gfCNCPoint2[16840] = {X 155.3044, Y 59.7694, Z -3.0000, A 0.000, B 0.000, C 0.000 }
gfCNCPoint2[16841] = {X 155.2181, Y 58.9678, Z -3.0000, A 0.000, B 0.000, C 0.000 }
gfCNCPoint2[16842] = {X 155.2180, Y 58.0000, Z -3.0000, A 0.000, B 0.000, C 0.000 }
gfCNCPoint2[16843] = {X 155.3203, Y 57.0921, Z -3.0000, A 0.000, B 0.000, C 0.000 }
gfCNCPoint2[16844] = {X 155.6220, Y 56.2298, Z -3.0000, A 0.000, B 0.000, C 0.000 }
gfCNCPoint2[16845] = {X 156.1081, Y 55.4562, Z -3.0000, A 0.000, B 0.000, C 0.000 }
gfCNCPoint2[16846] = {X 156.7541, Y 54.8101, Z -3.0000, A 0.000, B 0.000, C 0.000 }
gfCNCPoint2[16847] = {X 157.5277, Y 54.3240, Z -3.0000, A 0.000, B 0.000, C 0.000 }
gfCNCPoint2[16848] = {X 158.3901, Y 54.0223, Z -3.0000, A 0.000, B 0.000, C 0.000 }
gfCNCPoint2[16849] = {X 159.2980, Y 53.9200, Z -3.0000, A 0.000, B 0.000, C 0.000 }
gfCNCPoint2[16850] = {X 178.5335, Y 53.9200, Z -3.0000, A 0.000, B 0.000, C 0.000 }
gfCNCPoint2[16851] = {X 179.4414, Y 54.0223, Z -3.0000, A 0.000, B 0.000, C 0.000 }
gfCNCPoint2[16852] = {X 180.3037, Y 54.3240, Z -3.0000, A 0.000, B 0.000, C 0.000 }
gfCNCPoint2[16853] = {X 181.0773, Y 54.8101, Z -3.0000, A 0.000, B 0.000, C 0.000 }
gfCNCPoint2[16854] = {X 181.7234, Y 55.4562, Z -3.0000, A 0.000, B 0.000, C 0.000 }
gfCNCPoint2[16855] = {X 182.2095, Y 56.2298, Z -3.0000, A 0.000, B 0.000, C 0.000 }
gfCNCPoint2[16856] = {X 182.5112, Y 57.0921, Z -3.0000, A 0.000, B 0.000, C 0.000 }
gfCNCPoint2[16857] = {X 182.6135, Y 58.0000, Z -3.0000, A 0.000, B 0.000, C 0.000 }
gfCNCPoint2[16858] = {X 182.6135, Y 58.9342, Z -3.0000, A 0.000, B 0.000, C 0.000 }
gfCNCPoint2[16859] = {X 182.5334, Y 59.7385, Z -3.0000, A 0.000, B 0.000, C 0.000 }
gfCNCPoint2[16860] = {X 182.2963, Y 60.5113, Z -3.0000, A 0.000, B 0.000, C 0.000 }
gfCNCPoint2[16861] = {X 181.9116, Y 61.2221, Z -3.0000, A 0.000, B 0.000, C 0.000 }
gfCNCPoint2[16862] = {X 209.3010, Y 91.1161, Z -3.0000, A 0.000, B 0.000, C 0.000 }
gfCNCPoint2[16863] = {X 209.9711, Y 91.7959, Z -3.0000, A 0.000, B 0.000, C 0.000 }
gfCNCPoint2[16864] = {X 210.6888, Y 92.4252, Z -3.0000, A 0.000, B 0.000, C 0.000 }
gfCNCPoint2[16865] = {X 211.0137, Y 92.6303, Z -3.0000, A 0.000, B 0.000, C 0.000 }
gfCNCPoint2[16866] = {X 211.3781, Y 92.7521, Z -3.0000, A 0.000, B 0.000, C 0.000 }
gfCNCPoint2[16867] = {X 213.3970, Y 93.0670, Z -3.0000, A 0.000, B 0.000, C 0.000 }
gfCNCPoint2[16868] = {X 214.4547, Y 92.9770, Z -3.0000, A 0.000, B 0.000, C 0.000 }
gfCNCPoint2[16869] = {X 215.5145, Y 92.9161, Z -3.0000, A 0.000, B 0.000, C 0.000 }
gfCNCPoint2[16870] = {X 216.2276, Y 92.8376, Z -3.0000, A 0.000, B 0.000, C 0.000 }
gfCNCPoint2[16871] = {X 216.9142, Y 92.6297, Z -3.0000, A 0.000, B 0.000, C 0.000 }
gfCNCPoint2[16872] = {X 217.5510, Y 92.2995, Z -3.0000, A 0.000, B 0.000, C 0.000 }
gfCNCPoint2[16873] = {X 223.0910, Y 88.7242, Z -3.0000, A 0.000, B 0.000, C 0.000 }
gfCNCPoint2[16874] = {X 246.3547, Y 73.8481, Z -3.0000, A 0.000, B 0.000, C 0.000 }
gfCNCPoint2[16875] = {X 221.7196, Y 64.1802, Z -3.0000, A 0.000, B 0.000, C 0.000 }
gfCNCPoint2[16876] = {X 219.9262, Y 63.5800, Z -3.0000, A 0.000, B 0.000, C 0.000 }
gfCNCPoint2[16877] = {X 218.0758, Y 63.1888, Z -3.0000, A 0.000, B 0.000, C 0.000 }
gfCNCPoint2[16878] = {X 216.1929, Y 63.0117, Z -3.0000, A 0.000, B 0.000, C 0.000 }
gfCNCPoint2[16879] = {X 215.3127, Y 62.8850, Z -3.0000, A 0.000, B 0.000, C 0.000 }
gfCNCPoint2[16880] = {X 214.4809, Y 62.5706, Z -3.0000, A 0.000, B 0.000, C 0.000 }
gfCNCPoint2[16881] = {X 213.7370, Y 62.0834, Z -3.0000, A 0.000, B 0.000, C 0.000 }
gfCNCPoint2[16882] = {X 213.1162, Y 61.4466, Z -3.0000, A 0.000, B 0.000, C 0.000 }
gfCNCPoint2[16883] = {X 212.6482, Y 60.6905, Z -3.0000, A 0.000, B 0.000, C 0.000 }
gfCNCPoint2[16884] = {X 212.3552, Y 59.8509, Z -3.0000, A 0.000, B 0.000, C 0.000 }
gfCNCPoint2[16885] = {X 212.2509, Y 58.9678, Z -3.0000, A 0.000, B 0.000, C 0.000 }
gfCNCPoint2[16886] = {X 212.2508, Y 58.0000, Z -3.0000, A 0.000, B 0.000, C 0.000 }
gfCNCPoint2[16887] = {X 212.3531, Y 57.0921, Z -3.0000, A 0.000, B 0.000, C 0.000 }
gfCNCPoint2[16888] = {X 212.6549, Y 56.2298, Z -3.0000, A 0.000, B 0.000, C 0.000 }
gfCNCPoint2[16889] = {X 213.1409, Y 55.4562, Z -3.0000, A 0.000, B 0.000, C 0.000 }
gfCNCPoint2[16890] = {X 213.7870, Y 54.8101, Z -3.0000, A 0.000, B 0.000, C 0.000 }
gfCNCPoint2[16891] = {X 214.5606, Y 54.3240, Z -3.0000, A 0.000, B 0.000, C 0.000 }
gfCNCPoint2[16892] = {X 215.4229, Y 54.0223, Z -3.0000, A 0.000, B 0.000, C 0.000 }
gfCNCPoint2[16893] = {X 216.3308, Y 53.9200, Z -3.0000, A 0.000, B 0.000, C 0.000 }
gfCNCPoint2[16894] = {X 237.2617, Y 53.9200, Z -3.0000, A 0.000, B 0.000, C 0.000 }
gfCNCPoint2[16895] = {X 238.1696, Y 54.0223, Z -3.0000, A 0.000, B 0.000, C 0.000 }
gfCNCPoint2[16896] = {X 239.0319, Y 54.3240, Z -3.0000, A 0.000, B 0.000, C 0.000 }
gfCNCPoint2[16897] = {X 239.8055, Y 54.8101, Z -3.0000, A 0.000, B 0.000, C 0.000 }
gfCNCPoint2[16898] = {X 240.4516, Y 55.4562, Z -3.0000, A 0.000, B 0.000, C 0.000 }
gfCNCPoint2[16899] = {X 240.9376, Y 56.2298, Z -3.0000, A 0.000, B 0.000, C 0.000 }
gfCNCPoint2[16900] = {X 241.2394, Y 57.0921, Z -3.0000, A 0.000, B 0.000, C 0.000 }
gfCNCPoint2[16901] = {X 241.3417, Y 58.0000, Z -3.0000, A 0.000, B 0.000, C 0.000 }
gfCNCPoint2[16902] = {X 241.3417, Y 58.3967, Z -3.0000, A 0.000, B 0.000, C 0.000 }
gfCNCPoint2[16903] = {X 247.4005, Y 60.7586, Z -3.0000, A 0.000, B 0.000, C 0.000 }
gfCNCPoint2[16904] = {X 275.8735, Y 72.0561, Z -3.0000, A 0.000, B 0.000, C 0.000 }
gfCNCPoint2[16905] = {X 275.8743, Y 62.9983, Z -3.0000, A 0.000, B 0.000, C 0.000 }
gfCNCPoint2[16906] = {X 275.7380, Y 62.9840, Z -3.0000, A 0.000, B 0.000, C 0.000 }
gfCNCPoint2[16907] = {X 275.6022, Y 62.9651, Z -3.0000, A 0.000, B 0.000, C 0.000 }
gfCNCPoint2[16908] = {X 274.6826, Y 62.7081, Z -3.0000, A 0.000, B 0.000, C 0.000 }
gfCNCPoint2[16909] = {X 273.8479, Y 62.2445, Z -3.0000, A 0.000, B 0.000, C 0.000 }
gfCNCPoint2[16910] = {X 273.1438, Y 61.5996, Z -3.0000, A 0.000, B 0.000, C 0.000 }
gfCNCPoint2[16911] = {X 272.6088, Y 60.8087, Z -3.0000, A 0.000, B 0.000, C 0.000 }
gfCNCPoint2[16912] = {X 272.2724, Y 59.9151, Z -3.0000, A 0.000, B 0.000, C 0.000 }
gfCNCPoint2[16913] = {X 272.1528, Y 58.9678, Z -3.0000, A 0.000, B 0.000, C 0.000 }
gfCNCPoint2[16914] = {X 272.1527, Y 58.0000, Z -3.0000, A 0.000, B 0.000, C 0.000 }
gfCNCPoint2[16915] = {X 272.2550, Y 57.0921, Z -3.0000, A 0.000, B 0.000, C 0.000 }
gfCNCPoint2[16916] = {X 272.5567, Y 56.2298, Z -3.0000, A 0.000, B 0.000, C 0.000 }
gfCNCPoint2[16917] = {X 273.0428, Y 55.4562, Z -3.0000, A 0.000, B 0.000, C 0.000 }
gfCNCPoint2[16918] = {X 273.6889, Y 54.8101, Z -3.0000, A 0.000, B 0.000, C 0.000 }
gfCNCPoint2[16919] = {X 274.4624, Y 54.3240, Z -3.0000, A 0.000, B 0.000, C 0.000 }
gfCNCPoint2[16920] = {X 275.3248, Y 54.0223, Z -3.0000, A 0.000, B 0.000, C 0.000 }
gfCNCPoint2[16921] = {X 276.2327, Y 53.9200, Z -3.0000, A 0.000, B 0.000, C 0.000 }
gfCNCPoint2[16922] = {X 292.7731, Y 53.9200, Z -3.0000, A 0.000, B 0.000, C 0.000 }
gfCNCPoint2[16923] = {X 293.6810, Y 54.0223, Z -3.0000, A 0.000, B 0.000, C 0.000 }
gfCNCPoint2[16924] = {X 294.5433, Y 54.3240, Z -3.0000, A 0.000, B 0.000, C 0.000 }
gfCNCPoint2[16925] = {X 295.3169, Y 54.8101, Z -3.0000, A 0.000, B 0.000, C 0.000 }
gfCNCPoint2[16926] = {X 295.9630, Y 55.4562, Z -3.0000, A 0.000, B 0.000, C 0.000 }
gfCNCPoint2[16927] = {X 296.4490, Y 56.2298, Z -3.0000, A 0.000, B 0.000, C 0.000 }
gfCNCPoint2[16928] = {X 296.7508, Y 57.0921, Z -3.0000, A 0.000, B 0.000, C 0.000 }
gfCNCPoint2[16929] = {X 296.8531, Y 58.0000, Z -3.0000, A 0.000, B 0.000, C 0.000 }
gfCNCPoint2[16930] = {X 296.8531, Y 58.9344, Z -3.0000, A 0.000, B 0.000, C 0.000 }
gfCNCPoint2[16931] = {X 296.7374, Y 59.8874, Z -3.0000, A 0.000, B 0.000, C 0.000 }
gfCNCPoint2[16932] = {X 296.4031, Y 60.7873, Z -3.0000, A 0.000, B 0.000, C 0.000 }
gfCNCPoint2[16933] = {X 295.8686, Y 61.5848, Z -3.0000, A 0.000, B 0.000, C 0.000 }
gfCNCPoint2[16934] = {X 295.1631, Y 62.2359, Z -3.0000, A 0.000, B 0.000, C 0.000 }
gfCNCPoint2[16935] = {X 294.3255, Y 62.7050, Z -3.0000, A 0.000, B 0.000, C 0.000 }
gfCNCPoint2[16936] = {X 293.4017, Y 62.9663, Z -3.0000, A 0.000, B 0.000, C 0.000 }
gfCNCPoint2[16937] = {X 293.2752, Y 62.9845, Z -3.0000, A 0.000, B 0.000, C 0.000 }
gfCNCPoint2[16938] = {X 293.1481, Y 62.9987, Z -3.0000, A 0.000, B 0.000, C 0.000 }
gfCNCPoint2[16939] = {X 293.1321, Y 63.1581, Z -3.0000, A 0.000, B 0.000, C 0.000 }
gfCNCPoint2[16940] = {X 293.1443, Y 92.9938, Z -3.0000, A 0.000, B 0.000, C 0.000 }
gfCNCPoint2[16941] = {X 293.2728, Y 93.0085, Z -3.0000, A 0.000, B 0.000, C 0.000 }
gfCNCPoint2[16942] = {X 293.4007, Y 93.0272, Z -3.0000, A 0.000, B 0.000, C 0.000 }
gfCNCPoint2[16943] = {X 294.3242, Y 93.2911, Z -3.0000, A 0.000, B 0.000, C 0.000 }
gfCNCPoint2[16944] = {X 295.1614, Y 93.7620, Z -3.0000, A 0.000, B 0.000, C 0.000 }
gfCNCPoint2[16945] = {X 295.8665, Y 94.4142, Z -3.0000, A 0.000, B 0.000, C 0.000 }
gfCNCPoint2[16946] = {X 296.4011, Y 95.2122, Z -3.0000, A 0.000, B 0.000, C 0.000 }
gfCNCPoint2[16947] = {X 296.7360, Y 96.1124, Z -3.0000, A 0.000, B 0.000, C 0.000 }
gfCNCPoint2[16948] = {X 296.8531, Y 97.0657, Z -3.0000, A 0.000, B 0.000, C 0.000 }
gfCNCPoint2[16949] = {X 296.8531, Y 98.0000, Z -3.0000, A 0.000, B 0.000, C 0.000 }
gfCNCPoint2[16950] = {X 296.7508, Y 98.9079, Z -3.0000, A 0.000, B 0.000, C 0.000 }
gfCNCPoint2[16951] = {X 296.4490, Y 99.7702, Z -3.0000, A 0.000, B 0.000, C 0.000 }
gfCNCPoint2[16952] = {X 295.9630, Y 100.5438, Z -3.0000, A 0.000, B 0.000, C 0.000 }
gfCNCPoint2[16953] = {X 295.3169, Y 101.1899, Z -3.0000, A 0.000, B 0.000, C 0.000 }
gfCNCPoint2[16954] = {X 294.5433, Y 101.6760, Z -3.0000, A 0.000, B 0.000, C 0.000 }
gfCNCPoint2[16955] = {X 293.6810, Y 101.9777, Z -3.0000, A 0.000, B 0.000, C 0.000 }
gfCNCPoint2[16956] = {X 292.7731, Y 102.0800, Z -3.0000, A 0.000, B 0.000, C 0.000 }
gfCNCPoint2[16957] = {X 276.2327, Y 102.0800, Z -3.0000, A 0.000, B 0.000, C 0.000 }
gfCNCPoint2[16958] = {X 275.3248, Y 101.9777, Z -3.0000, A 0.000, B 0.000, C 0.000 }
gfCNCPoint2[16959] = {X 274.4624, Y 101.6760, Z -3.0000, A 0.000, B 0.000, C 0.000 }
gfCNCPoint2[16960] = {X 273.6889, Y 101.1899, Z -3.0000, A 0.000, B 0.000, C 0.000 }
gfCNCPoint2[16961] = {X 273.0428, Y 100.5438, Z -3.0000, A 0.000, B 0.000, C 0.000 }
gfCNCPoint2[16962] = {X 272.5567, Y 99.7702, Z -3.0000, A 0.000, B 0.000, C 0.000 }
gfCNCPoint2[16963] = {X 272.2550, Y 98.9079, Z -3.0000, A 0.000, B 0.000, C 0.000 }
gfCNCPoint2[16964] = {X 272.1527, Y 98.0000, Z -3.0000, A 0.000, B 0.000, C 0.000 }
gfCNCPoint2[16965] = {X 272.1527, Y 97.0659, Z -3.0000, A 0.000, B 0.000, C 0.000 }
gfCNCPoint2[16966] = {X 272.2437, Y 96.2088, Z -3.0000, A 0.000, B 0.000, C 0.000 }
gfCNCPoint2[16967] = {X 272.5128, Y 95.3899, Z -3.0000, A 0.000, B 0.000, C 0.000 }
gfCNCPoint2[16968] = {X 272.9480, Y 94.6458, Z -3.0000, A 0.000, B 0.000, C 0.000 }
gfCNCPoint2[16969] = {X 273.5297, Y 94.0097, Z -3.0000, A 0.000, B 0.000, C 0.000 }
gfCNCPoint2[16970] = {X 274.2321, Y 93.5101, Z -3.0000, A 0.000, B 0.000, C 0.000 }
gfCNCPoint2[16971] = {X 275.0238, Y 93.1692, Z -3.0000, A 0.000, B 0.000, C 0.000 }
gfCNCPoint2[16972] = {X 275.8694, Y 93.0021, Z -3.0000, A 0.000, B 0.000, C 0.000 }
gfCNCPoint2[16973] = {X 275.8694, Y 85.4313, Z -3.0000, A 0.000, B 0.000, C 0.000 }
gfCNCPoint2[16974] = {X 262.6143, Y 80.2353, Z -3.0000, A 0.000, B 0.000, C 0.000 }
gfCNCPoint2[16975] = {X 262.1471, Y 80.5294, Z -3.0000, A 0.000, B 0.000, C 0.000 }
gfCNCPoint2[16976] = {X 237.5552, Y 96.4582, Z -3.0000, A 0.000, B 0.000, C 0.000 }
gfCNCPoint2[16977] = {X 237.5598, Y 97.0656, Z -3.0000, A 0.000, B 0.000, C 0.000 }
gfCNCPoint2[16978] = {X 237.5598, Y 98.0000, Z -3.0000, A 0.000, B 0.000, C 0.000 }
gfCNCPoint2[16979] = {X 237.4575, Y 98.9079, Z -3.0000, A 0.000, B 0.000, C 0.000 }
gfCNCPoint2[16980] = {X 237.1557, Y 99.7702, Z -3.0000, A 0.000, B 0.000, C 0.000 }
gfCNCPoint2[16981] = {X 236.6697, Y 100.5438, Z -3.0000, A 0.000, B 0.000, C 0.000 }
gfCNCPoint2[16982] = {X 236.0236, Y 101.1899, Z -3.0000, A 0.000, B 0.000, C 0.000 }
gfCNCPoint2[16983] = {X 235.2500, Y 101.6760, Z -3.0000, A 0.000, B 0.000, C 0.000 }
gfCNCPoint2[16984] = {X 234.3877, Y 101.9777, Z -3.0000, A 0.000, B 0.000, C 0.000 }
gfCNCPoint2[16985] = {X 233.4798, Y 102.0800, Z -3.0000, A 0.000, B 0.000, C 0.000 }
gfCNCPoint2[16986] = {X 214.1790, Y 102.0800, Z -3.0000, A 0.000, B 0.000, C 0.000 }
gfCNCPoint2[16987] = {X 213.7860, Y 102.0610, Z -3.0000, A 0.000, B 0.000, C 0.000 }
gfCNCPoint2[16988] = {X 213.3966, Y 102.0043, Z -3.0000, A 0.000, B 0.000, C 0.000 }
gfCNCPoint2[16989] = {X 213.0072, Y 102.0610, Z -3.0000, A 0.000, B 0.000, C 0.000 }
gfCNCPoint2[16990] = {X 212.6141, Y 102.0800, Z -3.0000, A 0.000, B 0.000, C 0.000 }
gfCNCPoint2[16991] = {X 194.9870, Y 102.0800, Z -3.0000, A 0.000, B 0.000, C 0.000 }
gfCNCPoint2[16992] = {X 194.0791, Y 101.9777, Z -3.0000, A 0.000, B 0.000, C 0.000 }
gfCNCPoint2[16993] = {X 193.2167, Y 101.6760, Z -3.0000, A 0.000, B 0.000, C 0.000 }
gfCNCPoint2[16994] = {X 192.4431, Y 101.1899, Z -3.0000, A 0.000, B 0.000, C 0.000 }
gfCNCPoint2[16995] = {X 191.7971, Y 100.5438, Z -3.0000, A 0.000, B 0.000, C 0.000 }
gfCNCPoint2[16996] = {X 191.3110, Y 99.7702, Z -3.0000, A 0.000, B 0.000, C 0.000 }
gfCNCPoint2[16997] = {X 191.0093, Y 98.9079, Z -3.0000, A 0.000, B 0.000, C 0.000 }
gfCNCPoint2[16998] = {X 190.9070, Y 98.0000, Z -3.0000, A 0.000, B 0.000, C 0.000 }
gfCNCPoint2[16999] = {X 190.9070, Y 97.0659, Z -3.0000, A 0.000, B 0.000, C 0.000 }
gfCNCPoint2[17000] = {X 191.0022, Y 96.1894, Z -3.0000, A 0.000, B 0.000, C 0.000 }
gfCNCPoint2[17001] = {X 191.2835, Y 95.3539, Z -3.0000, A 0.000, B 0.000, C 0.000 }
gfCNCPoint2[17002] = {X 191.7378, Y 94.5983, Z -3.0000, A 0.000, B 0.000, C 0.000 }
gfCNCPoint2[17003] = {X 191.8199, Y 94.4938, Z -3.0000, A 0.000, B 0.000, C 0.000 }
gfCNCPoint2[17004] = {X 191.9053, Y 94.3920, Z -3.0000, A 0.000, B 0.000, C 0.000 }
gfCNCPoint2[17005] = {X 188.6703, Y 90.8602, Z -3.0000, A 0.000, B 0.000, C 0.000 }
gfCNCPoint2[17006] = {X 149.9831, Y 90.8602, Z -3.0000, A 0.000, B 0.000, C 0.000 }
gfCNCPoint2[17007] = {X 146.8263, Y 94.3576, Z -3.0000, A 0.000, B 0.000, C 0.000 }
gfCNCPoint2[17008] = {X 147.3862, Y 95.1680, Z -3.0000, A 0.000, B 0.000, C 0.000 }
gfCNCPoint2[17009] = {X 147.7372, Y 96.0884, Z -3.0000, A 0.000, B 0.000, C 0.000 }
gfCNCPoint2[17010] = {X 147.8591, Y 97.0658, Z -3.0000, A 0.000, B 0.000, C 0.000 }
gfCNCPoint2[17011] = {X 147.8591, Y 98.0000, Z -3.0000, A 0.000, B 0.000, C 0.000 }
gfCNCPoint2[17012] = {X 147.7568, Y 98.9079, Z -3.0000, A 0.000, B 0.000, C 0.000 }
gfCNCPoint2[17013] = {X 147.4551, Y 99.7702, Z -3.0000, A 0.000, B 0.000, C 0.000 }
gfCNCPoint2[17014] = {X 146.9690, Y 100.5438, Z -3.0000, A 0.000, B 0.000, C 0.000 }
gfCNCPoint2[17015] = {X 146.3229, Y 101.1899, Z -3.0000, A 0.000, B 0.000, C 0.000 }
gfCNCPoint2[17016] = {X 145.5494, Y 101.6760, Z -3.0000, A 0.000, B 0.000, C 0.000 }
gfCNCPoint2[17017] = {X 144.6870, Y 101.9777, Z -3.0000, A 0.000, B 0.000, C 0.000 }
gfCNCPoint2[17018] = {X 143.7791, Y 102.0800, Z -3.0000, A 0.000, B 0.000, C 0.000 }
gfCNCPoint2[17019] = {X 125.0000, Y 102.0800, Z -3.0000, A 0.000, B 0.000, C 0.000 }
gfCNCPoint2[17020] = {X 124.0921, Y 101.9777, Z -3.0000, A 0.000, B 0.000, C 0.000 }
gfCNCPoint2[17021] = {X 123.2298, Y 101.6760, Z -3.0000, A 0.000, B 0.000, C 0.000 }
gfCNCPoint2[17022] = {X 122.4562, Y 101.1899, Z -3.0000, A 0.000, B 0.000, C 0.000 }
gfCNCPoint2[17023] = {X 121.8101, Y 100.5438, Z -3.0000, A 0.000, B 0.000, C 0.000 }
gfCNCPoint2[17024] = {X 121.3240, Y 99.7702, Z -3.0000, A 0.000, B 0.000, C 0.000 }
gfCNCPoint2[17025] = {X 121.0223, Y 98.9079, Z -3.0000, A 0.000, B 0.000, C 0.000 }
gfCNCPoint2[17026] = {X 120.9200, Y 98.0000, Z -3.0000, A 0.000, B 0.000, C 0.000 }
gfCNCPoint2[17027] = {X 120.9200, Y 97.0659, Z -3.0000, A 0.000, B 0.000, C 0.000 }
gfCNCPoint2[17028] = {X 121.0194, Y 96.1709, Z -3.0000, A 0.000, B 0.000, C 0.000 }
gfCNCPoint2[17029] = {X 121.3127, Y 95.3195, Z -3.0000, A 0.000, B 0.000, C 0.000 }
gfCNCPoint2[17030] = {X 121.7856, Y 94.5532, Z -3.0000, A 0.000, B 0.000, C 0.000 }
gfCNCPoint2[17031] = {X 122.4151, Y 93.9092, Z -3.0000, A 0.000, B 0.000, C 0.000 }
gfCNCPoint2[17032] = {X 123.1706, Y 93.4191, Z -3.0000, A 0.000, B 0.000, C 0.000 }
gfCNCPoint2[17033] = {X 124.0151, Y 93.1066, Z -3.0000, A 0.000, B 0.000, C 0.000 }
gfCNCPoint2[17034] = {X 124.9076, Y 92.9870, Z -3.0000, A 0.000, B 0.000, C 0.000 }
gfCNCPoint2[17035] = {X 124.9313, Y 92.9716, Z -3.0000, A 0.000, B 0.000, C 0.000 }
gfCNCPoint2[17036] = {X 124.9632, Y 92.9595, Z -3.0000, A 0.000, B 0.000, C 0.000 }
gfCNCPoint2[17037] = {X 125.4828, Y 92.8824, Z -3.0000, A 0.000, B 0.000, C 0.000 }
gfCNCPoint2[17038] = {X 126.3569, Y 92.7337, Z -3.0000, A 0.000, B 0.000, C 0.000 }
gfCNCPoint2[17039] = {X 127.2186, Y 92.5246, Z -3.0000, A 0.000, B 0.000, C 0.000 }
gfCNCPoint2[17040] = {X 128.4717, Y 91.3464, Z -3.0000, A 0.000, B 0.000, C 0.000 }
gfCNCPoint2[17041] = {X 129.6579, Y 90.1009, Z -3.0000, A 0.000, B 0.000, C 0.000 }
gfCNCPoint2[17042] = {X 140.8578, Y 77.8019, Z -3.0000, A 0.000, B 0.000, C 0.000 }
gfCNCPoint2[17043] = {X 137.8977, Y 75.1063, Z -3.0000, A 0.000, B 0.000, C 0.000 }
gfCNCPoint2[17044] = {X 137.8982, Y 75.1058, Z -3.0000, A 0.000, B 0.000, C 0.000 }
gfCNCPoint2[17045] = {X 140.9144, Y 77.8534, Z -3.0000, A 0.000, B 0.000, C 0.000 }
gfCNCPoint2[17046] = {X 156.0375, Y 61.2513, Z -3.0000, A 0.000, B 0.000, C 0.000 }
gfCNCPoint2[17047] = {X 155.6325, Y 60.5356, Z -3.0000, A 0.000, B 0.000, C 0.000 }
gfCNCPoint2[17048] = {X 155.3825, Y 59.7521, Z -3.0000, A 0.000, B 0.000, C 0.000 }
gfCNCPoint2[17049] = {X 155.2980, Y 58.9340, Z -3.0000, A 0.000, B 0.000, C 0.000 }
gfCNCPoint2[17050] = {X 155.2980, Y 58.0000, Z -3.0000, A 0.000, B 0.000, C 0.000 }
gfCNCPoint2[17051] = {X 155.3982, Y 57.1099, Z -3.0000, A 0.000, B 0.000, C 0.000 }
gfCNCPoint2[17052] = {X 155.6941, Y 56.2645, Z -3.0000, A 0.000, B 0.000, C 0.000 }
gfCNCPoint2[17053] = {X 156.1706, Y 55.5060, Z -3.0000, A 0.000, B 0.000, C 0.000 }
gfCNCPoint2[17054] = {X 156.8040, Y 54.8727, Z -3.0000, A 0.000, B 0.000, C 0.000 }
gfCNCPoint2[17055] = {X 157.5624, Y 54.3961, Z -3.0000, A 0.000, B 0.000, C 0.000 }
gfCNCPoint2[17056] = {X 158.4079, Y 54.1003, Z -3.0000, A 0.000, B 0.000, C 0.000 }
gfCNCPoint2[17057] = {X 159.2980, Y 54.0000, Z -3.0000, A 0.000, B 0.000, C 0.000 }
gfCNCPoint2[17058] = {X 178.5335, Y 54.0000, Z -3.0000, A 0.000, B 0.000, C 0.000 }
gfCNCPoint2[17059] = {X 179.4236, Y 54.1003, Z -3.0000, A 0.000, B 0.000, C 0.000 }
gfCNCPoint2[17060] = {X 180.2690, Y 54.3961, Z -3.0000, A 0.000, B 0.000, C 0.000 }
gfCNCPoint2[17061] = {X 181.0275, Y 54.8727, Z -3.0000, A 0.000, B 0.000, C 0.000 }
gfCNCPoint2[17062] = {X 181.6608, Y 55.5060, Z -3.0000, A 0.000, B 0.000, C 0.000 }
gfCNCPoint2[17063] = {X 182.1374, Y 56.2645, Z -3.0000, A 0.000, B 0.000, C 0.000 }
gfCNCPoint2[17064] = {X 182.4332, Y 57.1099, Z -3.0000, A 0.000, B 0.000, C 0.000 }
gfCNCPoint2[17065] = {X 182.5335, Y 58.0000, Z -3.0000, A 0.000, B 0.000, C 0.000 }
gfCNCPoint2[17066] = {X 182.5334, Y 58.9671, Z -3.0000, A 0.000, B 0.000, C 0.000 }
gfCNCPoint2[17067] = {X 182.4463, Y 59.7648, Z -3.0000, A 0.000, B 0.000, C 0.000 }
gfCNCPoint2[17068] = {X 182.2017, Y 60.5291, Z -3.0000, A 0.000, B 0.000, C 0.000 }
gfCNCPoint2[17069] = {X 181.8095, Y 61.2292, Z -3.0000, A 0.000, B 0.000, C 0.000 }
gfCNCPoint2[17070] = {X 209.2420, Y 91.1701, Z -3.0000, A 0.000, B 0.000, C 0.000 }
gfCNCPoint2[17071] = {X 209.9162, Y 91.8541, Z -3.0000, A 0.000, B 0.000, C 0.000 }
gfCNCPoint2[17072] = {X 210.6383, Y 92.4872, Z -3.0000, A 0.000, B 0.000, C 0.000 }
gfCNCPoint2[17073] = {X 210.9795, Y 92.7026, Z -3.0000, A 0.000, B 0.000, C 0.000 }
gfCNCPoint2[17074] = {X 211.3621, Y 92.8305, Z -3.0000, A 0.000, B 0.000, C 0.000 }
gfCNCPoint2[17075] = {X 212.0545, Y 92.9785, Z -3.0000, A 0.000, B 0.000, C 0.000 }
gfCNCPoint2[17076] = {X 213.3960, Y 93.1475, Z -3.0000, A 0.000, B 0.000, C 0.000 }
gfCNCPoint2[17077] = {X 214.4554, Y 93.0572, Z -3.0000, A 0.000, B 0.000, C 0.000 }
gfCNCPoint2[17078] = {X 215.5170, Y 92.9961, Z -3.0000, A 0.000, B 0.000, C 0.000 }
gfCNCPoint2[17079] = {X 216.2444, Y 92.9159, Z -3.0000, A 0.000, B 0.000, C 0.000 }
gfCNCPoint2[17080] = {X 216.9448, Y 92.7036, Z -3.0000, A 0.000, B 0.000, C 0.000 }
gfCNCPoint2[17081] = {X 217.5944, Y 92.3667, Z -3.0000, A 0.000, B 0.000, C 0.000 }
gfCNCPoint2[17082] = {X 223.1343, Y 88.7915, Z -3.0000, A 0.000, B 0.000, C 0.000 }
gfCNCPoint2[17083] = {X 246.5300, Y 73.8309, Z -3.0000, A 0.000, B 0.000, C 0.000 }
gfCNCPoint2[17084] = {X 221.7493, Y 64.1059, Z -3.0000, A 0.000, B 0.000, C 0.000 }
gfCNCPoint2[17085] = {X 219.9472, Y 63.5028, Z -3.0000, A 0.000, B 0.000, C 0.000 }
gfCNCPoint2[17086] = {X 218.0879, Y 63.1097, Z -3.0000, A 0.000, B 0.000, C 0.000 }
gfCNCPoint2[17087] = {X 216.1958, Y 62.9318, Z -3.0000, A 0.000, B 0.000, C 0.000 }
gfCNCPoint2[17088] = {X 215.3283, Y 62.8064, Z -3.0000, A 0.000, B 0.000, C 0.000 }
gfCNCPoint2[17089] = {X 214.5089, Y 62.4950, Z -3.0000, A 0.000, B 0.000, C 0.000 }
gfCNCPoint2[17090] = {X 213.7770, Y 62.0127, Z -3.0000, A 0.000, B 0.000, C 0.000 }
gfCNCPoint2[17091] = {X 213.1677, Y 61.3825, Z -3.0000, A 0.000, B 0.000, C 0.000 }
gfCNCPoint2[17092] = {X 212.7104, Y 60.6348, Z -3.0000, A 0.000, B 0.000, C 0.000 }
gfCNCPoint2[17093] = {X 212.4268, Y 59.8053, Z -3.0000, A 0.000, B 0.000, C 0.000 }
gfCNCPoint2[17094] = {X 212.3308, Y 58.9340, Z -3.0000, A 0.000, B 0.000, C 0.000 }
gfCNCPoint2[17095] = {X 212.3308, Y 58.0000, Z -3.0000, A 0.000, B 0.000, C 0.000 }
gfCNCPoint2[17096] = {X 212.4311, Y 57.1099, Z -3.0000, A 0.000, B 0.000, C 0.000 }
gfCNCPoint2[17097] = {X 212.7269, Y 56.2645, Z -3.0000, A 0.000, B 0.000, C 0.000 }
gfCNCPoint2[17098] = {X 213.2035, Y 55.5060, Z -3.0000, A 0.000, B 0.000, C 0.000 }
gfCNCPoint2[17099] = {X 213.8368, Y 54.8727, Z -3.0000, A 0.000, B 0.000, C 0.000 }
gfCNCPoint2[17100] = {X 214.5953, Y 54.3961, Z -3.0000, A 0.000, B 0.000, C 0.000 }
gfCNCPoint2[17101] = {X 215.4407, Y 54.1003, Z -3.0000, A 0.000, B 0.000, C 0.000 }
gfCNCPoint2[17102] = {X 216.3308, Y 54.0000, Z -3.0000, A 0.000, B 0.000, C 0.000 }
gfCNCPoint2[17103] = {X 237.2617, Y 54.0000, Z -3.0000, A 0.000, B 0.000, C 0.000 }
gfCNCPoint2[17104] = {X 238.1518, Y 54.1003, Z -3.0000, A 0.000, B 0.000, C 0.000 }
gfCNCPoint2[17105] = {X 238.9972, Y 54.3961, Z -3.0000, A 0.000, B 0.000, C 0.000 }
gfCNCPoint2[17106] = {X 239.7556, Y 54.8727, Z -3.0000, A 0.000, B 0.000, C 0.000 }
gfCNCPoint2[17107] = {X 240.3890, Y 55.5060, Z -3.0000, A 0.000, B 0.000, C 0.000 }
gfCNCPoint2[17108] = {X 240.8656, Y 56.2645, Z -3.0000, A 0.000, B 0.000, C 0.000 }
gfCNCPoint2[17109] = {X 241.1614, Y 57.1099, Z -3.0000, A 0.000, B 0.000, C 0.000 }
gfCNCPoint2[17110] = {X 241.2617, Y 58.0000, Z -3.0000, A 0.000, B 0.000, C 0.000 }
gfCNCPoint2[17111] = {X 241.2617, Y 58.4514, Z -3.0000, A 0.000, B 0.000, C 0.000 }
gfCNCPoint2[17112] = {X 247.3712, Y 60.8331, Z -3.0000, A 0.000, B 0.000, C 0.000 }
gfCNCPoint2[17113] = {X 275.9535, Y 72.1739, Z -3.0000, A 0.000, B 0.000, C 0.000 }
gfCNCPoint2[17114] = {X 275.9528, Y 63.0383, Z -3.0000, A 0.000, B 0.000, C 0.000 }
gfCNCPoint2[17115] = {X 275.9573, Y 62.9246, Z -3.0000, A 0.000, B 0.000, C 0.000 }
gfCNCPoint2[17116] = {X 275.7855, Y 62.9090, Z -3.0000, A 0.000, B 0.000, C 0.000 }
gfCNCPoint2[17117] = {X 275.6146, Y 62.8860, Z -3.0000, A 0.000, B 0.000, C 0.000 }
gfCNCPoint2[17118] = {X 274.7079, Y 62.6320, Z -3.0000, A 0.000, B 0.000, C 0.000 }
gfCNCPoint2[17119] = {X 273.8857, Y 62.1732, Z -3.0000, A 0.000, B 0.000, C 0.000 }
gfCNCPoint2[17120] = {X 273.1936, Y 61.5348, Z -3.0000, A 0.000, B 0.000, C 0.000 }
gfCNCPoint2[17121] = {X 272.6698, Y 60.7523, Z -3.0000, A 0.000, B 0.000, C 0.000 }
gfCNCPoint2[17122] = {X 272.3435, Y 59.8691, Z -3.0000, A 0.000, B 0.000, C 0.000 }
gfCNCPoint2[17123] = {X 272.2327, Y 58.9340, Z -3.0000, A 0.000, B 0.000, C 0.000 }
gfCNCPoint2[17124] = {X 272.2327, Y 58.0000, Z -3.0000, A 0.000, B 0.000, C 0.000 }
gfCNCPoint2[17125] = {X 272.3330, Y 57.1099, Z -3.0000, A 0.000, B 0.000, C 0.000 }
gfCNCPoint2[17126] = {X 272.6288, Y 56.2645, Z -3.0000, A 0.000, B 0.000, C 0.000 }
gfCNCPoint2[17127] = {X 273.1054, Y 55.5060, Z -3.0000, A 0.000, B 0.000, C 0.000 }
gfCNCPoint2[17128] = {X 273.7387, Y 54.8727, Z -3.0000, A 0.000, B 0.000, C 0.000 }
gfCNCPoint2[17129] = {X 274.4972, Y 54.3961, Z -3.0000, A 0.000, B 0.000, C 0.000 }
gfCNCPoint2[17130] = {X 275.3426, Y 54.1003, Z -3.0000, A 0.000, B 0.000, C 0.000 }
gfCNCPoint2[17131] = {X 276.2327, Y 54.0000, Z -3.0000, A 0.000, B 0.000, C 0.000 }
gfCNCPoint2[17132] = {X 292.7731, Y 54.0000, Z -3.0000, A 0.000, B 0.000, C 0.000 }
gfCNCPoint2[17133] = {X 293.6632, Y 54.1003, Z -3.0000, A 0.000, B 0.000, C 0.000 }
gfCNCPoint2[17134] = {X 294.5086, Y 54.3961, Z -3.0000, A 0.000, B 0.000, C 0.000 }
gfCNCPoint2[17135] = {X 295.2670, Y 54.8727, Z -3.0000, A 0.000, B 0.000, C 0.000 }
gfCNCPoint2[17136] = {X 295.9004, Y 55.5060, Z -3.0000, A 0.000, B 0.000, C 0.000 }
gfCNCPoint2[17137] = {X 296.3770, Y 56.2645, Z -3.0000, A 0.000, B 0.000, C 0.000 }
gfCNCPoint2[17138] = {X 296.6728, Y 57.1099, Z -3.0000, A 0.000, B 0.000, C 0.000 }
gfCNCPoint2[17139] = {X 296.7731, Y 58.0000, Z -3.0000, A 0.000, B 0.000, C 0.000 }
gfCNCPoint2[17140] = {X 296.7731, Y 58.9341, Z -3.0000, A 0.000, B 0.000, C 0.000 }
gfCNCPoint2[17141] = {X 296.6597, Y 59.8685, Z -3.0000, A 0.000, B 0.000, C 0.000 }
gfCNCPoint2[17142] = {X 296.3319, Y 60.7509, Z -3.0000, A 0.000, B 0.000, C 0.000 }
gfCNCPoint2[17143] = {X 295.8078, Y 61.5328, Z -3.0000, A 0.000, B 0.000, C 0.000 }
gfCNCPoint2[17144] = {X 295.1161, Y 62.1712, Z -3.0000, A 0.000, B 0.000, C 0.000 }
gfCNCPoint2[17145] = {X 294.2948, Y 62.6311, Z -3.0000, A 0.000, B 0.000, C 0.000 }
gfCNCPoint2[17146] = {X 293.3891, Y 62.8873, Z -3.0000, A 0.000, B 0.000, C 0.000 }
gfCNCPoint2[17147] = {X 293.2325, Y 62.9091, Z -3.0000, A 0.000, B 0.000, C 0.000 }
gfCNCPoint2[17148] = {X 293.0752, Y 62.9248, Z -3.0000, A 0.000, B 0.000, C 0.000 }
gfCNCPoint2[17149] = {X 293.0521, Y 63.1540, Z -3.0000, A 0.000, B 0.000, C 0.000 }
gfCNCPoint2[17150] = {X 293.0521, Y 92.9237, Z -3.0000, A 0.000, B 0.000, C 0.000 }
gfCNCPoint2[17151] = {X 293.0752, Y 93.0678, Z -3.0000, A 0.000, B 0.000, C 0.000 }
gfCNCPoint2[17152] = {X 293.2319, Y 93.0839, Z -3.0000, A 0.000, B 0.000, C 0.000 }
gfCNCPoint2[17153] = {X 293.3879, Y 93.1062, Z -3.0000, A 0.000, B 0.000, C 0.000 }
gfCNCPoint2[17154] = {X 294.2934, Y 93.3649, Z -3.0000, A 0.000, B 0.000, C 0.000 }
gfCNCPoint2[17155] = {X 295.1143, Y 93.8267, Z -3.0000, A 0.000, B 0.000, C 0.000 }
gfCNCPoint2[17156] = {X 295.8057, Y 94.4662, Z -3.0000, A 0.000, B 0.000, C 0.000 }
gfCNCPoint2[17157] = {X 296.3299, Y 95.2486, Z -3.0000, A 0.000, B 0.000, C 0.000 }
gfCNCPoint2[17158] = {X 296.6583, Y 96.1313, Z -3.0000, A 0.000, B 0.000, C 0.000 }
gfCNCPoint2[17159] = {X 296.7731, Y 97.0661, Z -3.0000, A 0.000, B 0.000, C 0.000 }
gfCNCPoint2[17160] = {X 296.7731, Y 98.0000, Z -3.0000, A 0.000, B 0.000, C 0.000 }
gfCNCPoint2[17161] = {X 296.6728, Y 98.8901, Z -3.0000, A 0.000, B 0.000, C 0.000 }
gfCNCPoint2[17162] = {X 296.3770, Y 99.7355, Z -3.0000, A 0.000, B 0.000, C 0.000 }
gfCNCPoint2[17163] = {X 295.9004, Y 100.4940, Z -3.0000, A 0.000, B 0.000, C 0.000 }
gfCNCPoint2[17164] = {X 295.2670, Y 101.1273, Z -3.0000, A 0.000, B 0.000, C 0.000 }
gfCNCPoint2[17165] = {X 294.5086, Y 101.6039, Z -3.0000, A 0.000, B 0.000, C 0.000 }
gfCNCPoint2[17166] = {X 293.6632, Y 101.8997, Z -3.0000, A 0.000, B 0.000, C 0.000 }
gfCNCPoint2[17167] = {X 292.7731, Y 102.0000, Z -3.0000, A 0.000, B 0.000, C 0.000 }
gfCNCPoint2[17168] = {X 276.2327, Y 102.0000, Z -3.0000, A 0.000, B 0.000, C 0.000 }
gfCNCPoint2[17169] = {X 275.3426, Y 101.8997, Z -3.0000, A 0.000, B 0.000, C 0.000 }
gfCNCPoint2[17170] = {X 274.4972, Y 101.6039, Z -3.0000, A 0.000, B 0.000, C 0.000 }
gfCNCPoint2[17171] = {X 273.7387, Y 101.1273, Z -3.0000, A 0.000, B 0.000, C 0.000 }
gfCNCPoint2[17172] = {X 273.1054, Y 100.4940, Z -3.0000, A 0.000, B 0.000, C 0.000 }
gfCNCPoint2[17173] = {X 272.6288, Y 99.7355, Z -3.0000, A 0.000, B 0.000, C 0.000 }
gfCNCPoint2[17174] = {X 272.3330, Y 98.8901, Z -3.0000, A 0.000, B 0.000, C 0.000 }
gfCNCPoint2[17175] = {X 272.2327, Y 98.0000, Z -3.0000, A 0.000, B 0.000, C 0.000 }
gfCNCPoint2[17176] = {X 272.2329, Y 97.0232, Z -3.0000, A 0.000, B 0.000, C 0.000 }
gfCNCPoint2[17177] = {X 272.3321, Y 96.1797, Z -3.0000, A 0.000, B 0.000, C 0.000 }
gfCNCPoint2[17178] = {X 272.6072, Y 95.3761, Z -3.0000, A 0.000, B 0.000, C 0.000 }
gfCNCPoint2[17179] = {X 273.0457, Y 94.6486, Z -3.0000, A 0.000, B 0.000, C 0.000 }
gfCNCPoint2[17180] = {X 273.6280, Y 94.0302, Z -3.0000, A 0.000, B 0.000, C 0.000 }
gfCNCPoint2[17181] = {X 274.3277, Y 93.5487, Z -3.0000, A 0.000, B 0.000, C 0.000 }
gfCNCPoint2[17182] = {X 275.1133, Y 93.2258, Z -3.0000, A 0.000, B 0.000, C 0.000 }
gfCNCPoint2[17183] = {X 275.9494, Y 93.0760, Z -3.0000, A 0.000, B 0.000, C 0.000 }
gfCNCPoint2[17184] = {X 275.9494, Y 85.3767, Z -3.0000, A 0.000, B 0.000, C 0.000 }
gfCNCPoint2[17185] = {X 262.6059, Y 80.1460, Z -3.0000, A 0.000, B 0.000, C 0.000 }
gfCNCPoint2[17186] = {X 262.1040, Y 80.4620, Z -3.0000, A 0.000, B 0.000, C 0.000 }
gfCNCPoint2[17187] = {X 237.4749, Y 96.4149, Z -3.0000, A 0.000, B 0.000, C 0.000 }
gfCNCPoint2[17188] = {X 237.4798, Y 97.0659, Z -3.0000, A 0.000, B 0.000, C 0.000 }
gfCNCPoint2[17189] = {X 237.4798, Y 98.0000, Z -3.0000, A 0.000, B 0.000, C 0.000 }
gfCNCPoint2[17190] = {X 237.3795, Y 98.8901, Z -3.0000, A 0.000, B 0.000, C 0.000 }
gfCNCPoint2[17191] = {X 237.0837, Y 99.7355, Z -3.0000, A 0.000, B 0.000, C 0.000 }
gfCNCPoint2[17192] = {X 236.6071, Y 100.4940, Z -3.0000, A 0.000, B 0.000, C 0.000 }
gfCNCPoint2[17193] = {X 235.9737, Y 101.1273, Z -3.0000, A 0.000, B 0.000, C 0.000 }
gfCNCPoint2[17194] = {X 235.2153, Y 101.6039, Z -3.0000, A 0.000, B 0.000, C 0.000 }
gfCNCPoint2[17195] = {X 234.3699, Y 101.8997, Z -3.0000, A 0.000, B 0.000, C 0.000 }
gfCNCPoint2[17196] = {X 233.4798, Y 102.0000, Z -3.0000, A 0.000, B 0.000, C 0.000 }
gfCNCPoint2[17197] = {X 214.1790, Y 102.0000, Z -3.0000, A 0.000, B 0.000, C 0.000 }
gfCNCPoint2[17198] = {X 213.7859, Y 101.9806, Z -3.0000, A 0.000, B 0.000, C 0.000 }
gfCNCPoint2[17199] = {X 213.3966, Y 101.9227, Z -3.0000, A 0.000, B 0.000, C 0.000 }
gfCNCPoint2[17200] = {X 213.0072, Y 101.9806, Z -3.0000, A 0.000, B 0.000, C 0.000 }
gfCNCPoint2[17201] = {X 212.6141, Y 102.0000, Z -3.0000, A 0.000, B 0.000, C 0.000 }
gfCNCPoint2[17202] = {X 194.9870, Y 102.0000, Z -3.0000, A 0.000, B 0.000, C 0.000 }
gfCNCPoint2[17203] = {X 194.0969, Y 101.8997, Z -3.0000, A 0.000, B 0.000, C 0.000 }
gfCNCPoint2[17204] = {X 193.2514, Y 101.6039, Z -3.0000, A 0.000, B 0.000, C 0.000 }
gfCNCPoint2[17205] = {X 192.4930, Y 101.1273, Z -3.0000, A 0.000, B 0.000, C 0.000 }
gfCNCPoint2[17206] = {X 191.8596, Y 100.4940, Z -3.0000, A 0.000, B 0.000, C 0.000 }
gfCNCPoint2[17207] = {X 191.3831, Y 99.7355, Z -3.0000, A 0.000, B 0.000, C 0.000 }
gfCNCPoint2[17208] = {X 191.0872, Y 98.8901, Z -3.0000, A 0.000, B 0.000, C 0.000 }
gfCNCPoint2[17209] = {X 190.9870, Y 98.0000, Z -3.0000, A 0.000, B 0.000, C 0.000 }
gfCNCPoint2[17210] = {X 190.9870, Y 97.0659, Z -3.0000, A 0.000, B 0.000, C 0.000 }
gfCNCPoint2[17211] = {X 191.0804, Y 96.2066, Z -3.0000, A 0.000, B 0.000, C 0.000 }
gfCNCPoint2[17212] = {X 191.3562, Y 95.3874, Z -3.0000, A 0.000, B 0.000, C 0.000 }
gfCNCPoint2[17213] = {X 191.8015, Y 94.6466, Z -3.0000, A 0.000, B 0.000, C 0.000 }
gfCNCPoint2[17214] = {X 191.8852, Y 94.5402, Z -3.0000, A 0.000, B 0.000, C 0.000 }
gfCNCPoint2[17215] = {X 191.9725, Y 94.4367, Z -3.0000, A 0.000, B 0.000, C 0.000 }
gfCNCPoint2[17216] = {X 192.0151, Y 94.3934, Z -3.0000, A 0.000, B 0.000, C 0.000 }
gfCNCPoint2[17217] = {X 188.7055, Y 90.7802, Z -3.0000, A 0.000, B 0.000, C 0.000 }
gfCNCPoint2[17218] = {X 149.9476, Y 90.7802, Z -3.0000, A 0.000, B 0.000, C 0.000 }
gfCNCPoint2[17219] = {X 146.7186, Y 94.3576, Z -3.0000, A 0.000, B 0.000, C 0.000 }
gfCNCPoint2[17220] = {X 147.1683, Y 94.9489, Z -3.0000, A 0.000, B 0.000, C 0.000 }
gfCNCPoint2[17221] = {X 147.5018, Y 95.6128, Z -3.0000, A 0.000, B 0.000, C 0.000 }
gfCNCPoint2[17222] = {X 147.7077, Y 96.3266, Z -3.0000, A 0.000, B 0.000, C 0.000 }
gfCNCPoint2[17223] = {X 147.7791, Y 97.0661, Z -3.0000, A 0.000, B 0.000, C 0.000 }
gfCNCPoint2[17224] = {X 147.7791, Y 98.0000, Z -3.0000, A 0.000, B 0.000, C 0.000 }
gfCNCPoint2[17225] = {X 147.6788, Y 98.8901, Z -3.0000, A 0.000, B 0.000, C 0.000 }
gfCNCPoint2[17226] = {X 147.3830, Y 99.7355, Z -3.0000, A 0.000, B 0.000, C 0.000 }
gfCNCPoint2[17227] = {X 146.9064, Y 100.4940, Z -3.0000, A 0.000, B 0.000, C 0.000 }
gfCNCPoint2[17228] = {X 146.2731, Y 101.1273, Z -3.0000, A 0.000, B 0.000, C 0.000 }
gfCNCPoint2[17229] = {X 145.5146, Y 101.6039, Z -3.0000, A 0.000, B 0.000, C 0.000 }
gfCNCPoint2[17230] = {X 144.6692, Y 101.8997, Z -3.0000, A 0.000, B 0.000, C 0.000 }
gfCNCPoint2[17231] = {X 143.7791, Y 102.0000, Z -3.0000, A 0.000, B 0.000, C 0.000 }
gfCNCPoint2[17232] = {X 125.0000, Y 102.0000, Z -3.0000, A 0.000, B 0.000, C 0.000 }
gfCNCPoint2[17233] = {X 124.1099, Y 101.8997, Z -3.0000, A 0.000, B 0.000, C 0.000 }
gfCNCPoint2[17234] = {X 123.2645, Y 101.6039, Z -3.0000, A 0.000, B 0.000, C 0.000 }
gfCNCPoint2[17235] = {X 122.5060, Y 101.1273, Z -3.0000, A 0.000, B 0.000, C 0.000 }
gfCNCPoint2[17236] = {X 121.8727, Y 100.4940, Z -3.0000, A 0.000, B 0.000, C 0.000 }
gfCNCPoint2[17237] = {X 121.3961, Y 99.7355, Z -3.0000, A 0.000, B 0.000, C 0.000 }
gfCNCPoint2[17238] = {X 121.1003, Y 98.8901, Z -3.0000, A 0.000, B 0.000, C 0.000 }
gfCNCPoint2[17239] = {X 121.0000, Y 98.0000, Z -3.0000, A 0.000, B 0.000, C 0.000 }
gfCNCPoint2[17240] = {X 121.0000, Y 97.0659, Z -3.0000, A 0.000, B 0.000, C 0.000 }
gfCNCPoint2[17241] = {X 121.0981, Y 96.1853, Z -3.0000, A 0.000, B 0.000, C 0.000 }
gfCNCPoint2[17242] = {X 121.3877, Y 95.3479, Z -3.0000, A 0.000, B 0.000, C 0.000 }
gfCNCPoint2[17243] = {X 121.8546, Y 94.5948, Z -3.0000, A 0.000, B 0.000, C 0.000 }
gfCNCPoint2[17244] = {X 122.4758, Y 93.9629, Z -3.0000, A 0.000, B 0.000, C 0.000 }
gfCNCPoint2[17245] = {X 123.2209, Y 93.4834, Z -3.0000, A 0.000, B 0.000, C 0.000 }
gfCNCPoint2[17246] = {X 124.0533, Y 93.1796, Z -3.0000, A 0.000, B 0.000, C 0.000 }
gfCNCPoint2[17247] = {X 124.9321, Y 93.0665, Z -3.0000, A 0.000, B 0.000, C 0.000 }
gfCNCPoint2[17248] = {X 124.9749, Y 93.0387, Z -3.0000, A 0.000, B 0.000, C 0.000 }
gfCNCPoint2[17249] = {X 125.4940, Y 92.9616, Z -3.0000, A 0.000, B 0.000, C 0.000 }
gfCNCPoint2[17250] = {X 126.3824, Y 92.8101, Z -3.0000, A 0.000, B 0.000, C 0.000 }
gfCNCPoint2[17251] = {X 127.2579, Y 92.5967, Z -3.0000, A 0.000, B 0.000, C 0.000 }
gfCNCPoint2[17252] = {X 128.5215, Y 91.4097, Z -3.0000, A 0.000, B 0.000, C 0.000 }
gfCNCPoint2[17253] = {X 129.7173, Y 90.1544, Z -3.0000, A 0.000, B 0.000, C 0.000 }
gfCNCPoint2[17254] = {X 133.8038, Y 85.6592, Z -3.0000, A 0.000, B 0.000, C 0.000 }
gfCNCPoint2[17255] = {X 140.9144, Y 77.8534, Z -3.0000, A 0.000, B 0.000, C 0.000 }
gfCNCPoint2[17256] = {X 137.8982, Y 75.1058, Z -3.0000, A 0.000, B 0.000, C 0.000 }
gfCNCPoint2[17257] = {X 137.8982, Y 75.1058, Z 0.0000, A 0.000, B 0.000, C 0.000 }
gfCNCPoint2[17258] = {X 137.8982, Y 75.1058, Z 11.0000, A 0.000, B 0.000, C 0.000 }
gfCNCPoint2[17259] = {X 167.3809, Y 20.2812, Z 11.0000, A 0.000, B 0.000, C 0.000 }
gfCNCPoint2[17260] = {X 167.3809, Y 20.2812, Z 0.0000, A 0.000, B 0.000, C 0.000 }
gfCNCPoint2[17261] = {X 167.3809, Y 20.2812, Z -3.0000, A 0.000, B 0.000, C 0.000 }
gfCNCPoint2[17262] = {X 171.1581, Y 18.7388, Z -3.0000, A 0.000, B 0.000, C 0.000 }
gfCNCPoint2[17263] = {X 169.8405, Y 15.5121, Z -3.0000, A 0.000, B 0.000, C 0.000 }
gfCNCPoint2[17264] = {X 169.5912, Y 14.6607, Z -3.0000, A 0.000, B 0.000, C 0.000 }
gfCNCPoint2[17265] = {X 169.5212, Y 13.7764, Z -3.0000, A 0.000, B 0.000, C 0.000 }
gfCNCPoint2[17266] = {X 169.6332, Y 12.8964, Z -3.0000, A 0.000, B 0.000, C 0.000 }
gfCNCPoint2[17267] = {X 169.9226, Y 12.0578, Z -3.0000, A 0.000, B 0.000, C 0.000 }
gfCNCPoint2[17268] = {X 170.3773, Y 11.2960, Z -3.0000, A 0.000, B 0.000, C 0.000 }
gfCNCPoint2[17269] = {X 170.9779, Y 10.6432, Z -3.0000, A 0.000, B 0.000, C 0.000 }
gfCNCPoint2[17270] = {X 171.6992, Y 10.1268, Z -3.0000, A 0.000, B 0.000, C 0.000 }
gfCNCPoint2[17271] = {X 172.3295, Y 9.7674, Z -3.0000, A 0.000, B 0.000, C 0.000 }
gfCNCPoint2[17272] = {X 173.2114, Y 9.3960, Z -3.0000, A 0.000, B 0.000, C 0.000 }
gfCNCPoint2[17273] = {X 174.1534, Y 9.2278, Z -3.0000, A 0.000, B 0.000, C 0.000 }
gfCNCPoint2[17274] = {X 175.1093, Y 9.2711, Z -3.0000, A 0.000, B 0.000, C 0.000 }
gfCNCPoint2[17275] = {X 176.0323, Y 9.5238, Z -3.0000, A 0.000, B 0.000, C 0.000 }
gfCNCPoint2[17276] = {X 178.2250, Y 8.6012, Z -3.0000, A 0.000, B 0.000, C 0.000 }
gfCNCPoint2[17277] = {X 180.4989, Y 7.9025, Z -3.0000, A 0.000, B 0.000, C 0.000 }
gfCNCPoint2[17278] = {X 182.8314, Y 7.4348, Z -3.0000, A 0.000, B 0.000, C 0.000 }
gfCNCPoint2[17279] = {X 185.1990, Y 7.2027, Z -3.0000, A 0.000, B 0.000, C 0.000 }
gfCNCPoint2[17280] = {X 187.5779, Y 7.2085, Z -3.0000, A 0.000, B 0.000, C 0.000 }
gfCNCPoint2[17281] = {X 189.9442, Y 7.4523, Z -3.0000, A 0.000, B 0.000, C 0.000 }
gfCNCPoint2[17282] = {X 191.7015, Y 7.8138, Z -3.0000, A 0.000, B 0.000, C 0.000 }
gfCNCPoint2[17283] = {X 193.4123, Y 8.3538, Z -3.0000, A 0.000, B 0.000, C 0.000 }
gfCNCPoint2[17284] = {X 195.0587, Y 9.0665, Z -3.0000, A 0.000, B 0.000, C 0.000 }
gfCNCPoint2[17285] = {X 196.6232, Y 9.9445, Z -3.0000, A 0.000, B 0.000, C 0.000 }
gfCNCPoint2[17286] = {X 198.0893, Y 10.9785, Z -3.0000, A 0.000, B 0.000, C 0.000 }
gfCNCPoint2[17287] = {X 199.1489, Y 11.9219, Z -3.0000, A 0.000, B 0.000, C 0.000 }
gfCNCPoint2[17288] = {X 200.0998, Y 12.9747, Z -3.0000, A 0.000, B 0.000, C 0.000 }
gfCNCPoint2[17289] = {X 200.9308, Y 14.1245, Z -3.0000, A 0.000, B 0.000, C 0.000 }
gfCNCPoint2[17290] = {X 201.6321, Y 15.3578, Z -3.0000, A 0.000, B 0.000, C 0.000 }
gfCNCPoint2[17291] = {X 202.1953, Y 16.6598, Z -3.0000, A 0.000, B 0.000, C 0.000 }
gfCNCPoint2[17292] = {X 202.6696, Y 18.3162, Z -3.0000, A 0.000, B 0.000, C 0.000 }
gfCNCPoint2[17293] = {X 202.9510, Y 20.0160, Z -3.0000, A 0.000, B 0.000, C 0.000 }
gfCNCPoint2[17294] = {X 203.0360, Y 21.7368, Z -3.0000, A 0.000, B 0.000, C 0.000 }
gfCNCPoint2[17295] = {X 202.9235, Y 23.4560, Z -3.0000, A 0.000, B 0.000, C 0.000 }
gfCNCPoint2[17296] = {X 202.6148, Y 25.1510, Z -3.0000, A 0.000, B 0.000, C 0.000 }
gfCNCPoint2[17297] = {X 202.1730, Y 26.5971, Z -3.0000, A 0.000, B 0.000, C 0.000 }
gfCNCPoint2[17298] = {X 201.5483, Y 27.9741, Z -3.0000, A 0.000, B 0.000, C 0.000 }
gfCNCPoint2[17299] = {X 200.7511, Y 29.2590, Z -3.0000, A 0.000, B 0.000, C 0.000 }
gfCNCPoint2[17300] = {X 199.7947, Y 30.4302, Z -3.0000, A 0.000, B 0.000, C 0.000 }
gfCNCPoint2[17301] = {X 198.6952, Y 31.4682, Z -3.0000, A 0.000, B 0.000, C 0.000 }
gfCNCPoint2[17302] = {X 199.4967, Y 31.8094, Z -3.0000, A 0.000, B 0.000, C 0.000 }
gfCNCPoint2[17303] = {X 200.2134, Y 32.3045, Z -3.0000, A 0.000, B 0.000, C 0.000 }
gfCNCPoint2[17304] = {X 200.8163, Y 32.9332, Z -3.0000, A 0.000, B 0.000, C 0.000 }
gfCNCPoint2[17305] = {X 201.2808, Y 33.6702, Z -3.0000, A 0.000, B 0.000, C 0.000 }
gfCNCPoint2[17306] = {X 204.3222, Y 39.9530, Z -3.0000, A 0.000, B 0.000, C 0.000 }
gfCNCPoint2[17307] = {X 204.6427, Y 40.8622, Z -3.0000, A 0.000, B 0.000, C 0.000 }
gfCNCPoint2[17308] = {X 204.7537, Y 41.8197, Z -3.0000, A 0.000, B 0.000, C 0.000 }
gfCNCPoint2[17309] = {X 204.6496, Y 42.7781, Z -3.0000, A 0.000, B 0.000, C 0.000 }
gfCNCPoint2[17310] = {X 204.3355, Y 43.6895, Z -3.0000, A 0.000, B 0.000, C 0.000 }
gfCNCPoint2[17311] = {X 203.8272, Y 44.5085, Z -3.0000, A 0.000, B 0.000, C 0.000 }
gfCNCPoint2[17312] = {X 203.1499, Y 45.1945, Z -3.0000, A 0.000, B 0.000, C 0.000 }
gfCNCPoint2[17313] = {X 202.6135, Y 45.6281, Z -3.0000, A 0.000, B 0.000, C 0.000 }
gfCNCPoint2[17314] = {X 201.9089, Y 46.0916, Z -3.0000, A 0.000, B 0.000, C 0.000 }
gfCNCPoint2[17315] = {X 201.1277, Y 46.4098, Z -3.0000, A 0.000, B 0.000, C 0.000 }
gfCNCPoint2[17316] = {X 200.2998, Y 46.5707, Z -3.0000, A 0.000, B 0.000, C 0.000 }
gfCNCPoint2[17317] = {X 199.4564, Y 46.5682, Z -3.0000, A 0.000, B 0.000, C 0.000 }
gfCNCPoint2[17318] = {X 198.6294, Y 46.4025, Z -3.0000, A 0.000, B 0.000, C 0.000 }
gfCNCPoint2[17319] = {X 196.2990, Y 47.6048, Z -3.0000, A 0.000, B 0.000, C 0.000 }
gfCNCPoint2[17320] = {X 193.8686, Y 48.5894, Z -3.0000, A 0.000, B 0.000, C 0.000 }
gfCNCPoint2[17321] = {X 191.3585, Y 49.3481, Z -3.0000, A 0.000, B 0.000, C 0.000 }
gfCNCPoint2[17322] = {X 189.4154, Y 49.7418, Z -3.0000, A 0.000, B 0.000, C 0.000 }
gfCNCPoint2[17323] = {X 187.4453, Y 49.9641, Z -3.0000, A 0.000, B 0.000, C 0.000 }
gfCNCPoint2[17324] = {X 185.4634, Y 50.0133, Z -3.0000, A 0.000, B 0.000, C 0.000 }
gfCNCPoint2[17325] = {X 183.4847, Y 49.8889, Z -3.0000, A 0.000, B 0.000, C 0.000 }
gfCNCPoint2[17326] = {X 181.5245, Y 49.5920, Z -3.0000, A 0.000, B 0.000, C 0.000 }
gfCNCPoint2[17327] = {X 179.6380, Y 49.1205, Z -3.0000, A 0.000, B 0.000, C 0.000 }
gfCNCPoint2[17328] = {X 177.8176, Y 48.4370, Z -3.0000, A 0.000, B 0.000, C 0.000 }
gfCNCPoint2[17329] = {X 176.0869, Y 47.5506, Z -3.0000, A 0.000, B 0.000, C 0.000 }
gfCNCPoint2[17330] = {X 174.4686, Y 46.4726, Z -3.0000, A 0.000, B 0.000, C 0.000 }
gfCNCPoint2[17331] = {X 173.2358, Y 45.4321, Z -3.0000, A 0.000, B 0.000, C 0.000 }
gfCNCPoint2[17332] = {X 172.1388, Y 44.2494, Z -3.0000, A 0.000, B 0.000, C 0.000 }
gfCNCPoint2[17333] = {X 171.1939, Y 42.9420, Z -3.0000, A 0.000, B 0.000, C 0.000 }
gfCNCPoint2[17334] = {X 170.4150, Y 41.5293, Z -3.0000, A 0.000, B 0.000, C 0.000 }
gfCNCPoint2[17335] = {X 169.8138, Y 40.0324, Z -3.0000, A 0.000, B 0.000, C 0.000 }
gfCNCPoint2[17336] = {X 169.3992, Y 38.4735, Z -3.0000, A 0.000, B 0.000, C 0.000 }
gfCNCPoint2[17337] = {X 169.1773, Y 36.8757, Z -3.0000, A 0.000, B 0.000, C 0.000 }
gfCNCPoint2[17338] = {X 169.0931, Y 35.0417, Z -3.0000, A 0.000, B 0.000, C 0.000 }
gfCNCPoint2[17339] = {X 169.2393, Y 33.2117, Z -3.0000, A 0.000, B 0.000, C 0.000 }
gfCNCPoint2[17340] = {X 169.6134, Y 31.4144, Z -3.0000, A 0.000, B 0.000, C 0.000 }
gfCNCPoint2[17341] = {X 170.2096, Y 29.6780, Z -3.0000, A 0.000, B 0.000, C 0.000 }
gfCNCPoint2[17342] = {X 170.8486, Y 28.3710, Z -3.0000, A 0.000, B 0.000, C 0.000 }
gfCNCPoint2[17343] = {X 171.6565, Y 27.1611, Z -3.0000, A 0.000, B 0.000, C 0.000 }
gfCNCPoint2[17344] = {X 172.6189, Y 26.0700, Z -3.0000, A 0.000, B 0.000, C 0.000 }
gfCNCPoint2[17345] = {X 173.7184, Y 25.1173, Z -3.0000, A 0.000, B 0.000, C 0.000 }
gfCNCPoint2[17346] = {X 174.9354, Y 24.3201, Z -3.0000, A 0.000, B 0.000, C 0.000 }
gfCNCPoint2[17347] = {X 174.1526, Y 23.9325, Z -3.0000, A 0.000, B 0.000, C 0.000 }
gfCNCPoint2[17348] = {X 173.4638, Y 23.3953, Z -3.0000, A 0.000, B 0.000, C 0.000 }
gfCNCPoint2[17349] = {X 172.8972, Y 22.7306, Z -3.0000, A 0.000, B 0.000, C 0.000 }
gfCNCPoint2[17350] = {X 172.4758, Y 21.9655, Z -3.0000, A 0.000, B 0.000, C 0.000 }
gfCNCPoint2[17351] = {X 171.1581, Y 18.7388, Z -3.0000, A 0.000, B 0.000, C 0.000 }
gfCNCPoint2[17352] = {X 167.4550, Y 20.2510, Z -3.0000, A 0.000, B 0.000, C 0.000 }
gfCNCPoint2[17353] = {X 171.2322, Y 18.7085, Z -3.0000, A 0.000, B 0.000, C 0.000 }
gfCNCPoint2[17354] = {X 169.9145, Y 15.4818, Z -3.0000, A 0.000, B 0.000, C 0.000 }
gfCNCPoint2[17355] = {X 169.6699, Y 14.6462, Z -3.0000, A 0.000, B 0.000, C 0.000 }
gfCNCPoint2[17356] = {X 169.6011, Y 13.7783, Z -3.0000, A 0.000, B 0.000, C 0.000 }
gfCNCPoint2[17357] = {X 169.7111, Y 12.9146, Z -3.0000, A 0.000, B 0.000, C 0.000 }
gfCNCPoint2[17358] = {X 169.9952, Y 12.0915, Z -3.0000, A 0.000, B 0.000, C 0.000 }
gfCNCPoint2[17359] = {X 170.4414, Y 11.3439, Z -3.0000, A 0.000, B 0.000, C 0.000 }
gfCNCPoint2[17360] = {X 171.0309, Y 10.7031, Z -3.0000, A 0.000, B 0.000, C 0.000 }
gfCNCPoint2[17361] = {X 171.7389, Y 10.1963, Z -3.0000, A 0.000, B 0.000, C 0.000 }
gfCNCPoint2[17362] = {X 172.3689, Y 9.8371, Z -3.0000, A 0.000, B 0.000, C 0.000 }
gfCNCPoint2[17363] = {X 173.2427, Y 9.4701, Z -3.0000, A 0.000, B 0.000, C 0.000 }
gfCNCPoint2[17364] = {X 174.1763, Y 9.3065, Z -3.0000, A 0.000, B 0.000, C 0.000 }
gfCNCPoint2[17365] = {X 175.1229, Y 9.3543, Z -3.0000, A 0.000, B 0.000, C 0.000 }
gfCNCPoint2[17366] = {X 176.0352, Y 9.6112, Z -3.0000, A 0.000, B 0.000, C 0.000 }
gfCNCPoint2[17367] = {X 178.2246, Y 8.6864, Z -3.0000, A 0.000, B 0.000, C 0.000 }
gfCNCPoint2[17368] = {X 180.4958, Y 7.9858, Z -3.0000, A 0.000, B 0.000, C 0.000 }
gfCNCPoint2[17369] = {X 182.8258, Y 7.5165, Z -3.0000, A 0.000, B 0.000, C 0.000 }
gfCNCPoint2[17370] = {X 185.1910, Y 7.2832, Z -3.0000, A 0.000, B 0.000, C 0.000 }
gfCNCPoint2[17371] = {X 187.5678, Y 7.2881, Z -3.0000, A 0.000, B 0.000, C 0.000 }
gfCNCPoint2[17372] = {X 189.9321, Y 7.5314, Z -3.0000, A 0.000, B 0.000, C 0.000 }
gfCNCPoint2[17373] = {X 191.6813, Y 7.8912, Z -3.0000, A 0.000, B 0.000, C 0.000 }
gfCNCPoint2[17374] = {X 193.3843, Y 8.4287, Z -3.0000, A 0.000, B 0.000, C 0.000 }
gfCNCPoint2[17375] = {X 195.0232, Y 9.1382, Z -3.0000, A 0.000, B 0.000, C 0.000 }
gfCNCPoint2[17376] = {X 196.5805, Y 10.0122, Z -3.0000, A 0.000, B 0.000, C 0.000 }
gfCNCPoint2[17377] = {X 198.0399, Y 11.0414, Z -3.0000, A 0.000, B 0.000, C 0.000 }
gfCNCPoint2[17378] = {X 199.3397, Y 12.2309, Z -3.0000, A 0.000, B 0.000, C 0.000 }
gfCNCPoint2[17379] = {X 200.4662, Y 13.5854, Z -3.0000, A 0.000, B 0.000, C 0.000 }
gfCNCPoint2[17380] = {X 201.3989, Y 15.0802, Z -3.0000, A 0.000, B 0.000, C 0.000 }
gfCNCPoint2[17381] = {X 202.1203, Y 16.6876, Z -3.0000, A 0.000, B 0.000, C 0.000 }
gfCNCPoint2[17382] = {X 202.5918, Y 18.3349, Z -3.0000, A 0.000, B 0.000, C 0.000 }
gfCNCPoint2[17383] = {X 202.8716, Y 20.0254, Z -3.0000, A 0.000, B 0.000, C 0.000 }
gfCNCPoint2[17384] = {X 202.9560, Y 21.7368, Z -3.0000, A 0.000, B 0.000, C 0.000 }
gfCNCPoint2[17385] = {X 202.8440, Y 23.4466, Z -3.0000, A 0.000, B 0.000, C 0.000 }
gfCNCPoint2[17386] = {X 202.5370, Y 25.1324, Z -3.0000, A 0.000, B 0.000, C 0.000 }
gfCNCPoint2[17387] = {X 202.0875, Y 26.5970, Z -3.0000, A 0.000, B 0.000, C 0.000 }
gfCNCPoint2[17388] = {X 201.4491, Y 27.9897, Z -3.0000, A 0.000, B 0.000, C 0.000 }
gfCNCPoint2[17389] = {X 200.6329, Y 29.2862, Z -3.0000, A 0.000, B 0.000, C 0.000 }
gfCNCPoint2[17390] = {X 199.6532, Y 30.4639, Z -3.0000, A 0.000, B 0.000, C 0.000 }
gfCNCPoint2[17391] = {X 198.5269, Y 31.5025, Z -3.0000, A 0.000, B 0.000, C 0.000 }
gfCNCPoint2[17392] = {X 199.3585, Y 31.8263, Z -3.0000, A 0.000, B 0.000, C 0.000 }
gfCNCPoint2[17393] = {X 200.1038, Y 32.3171, Z -3.0000, A 0.000, B 0.000, C 0.000 }
gfCNCPoint2[17394] = {X 200.7300, Y 32.9529, Z -3.0000, A 0.000, B 0.000, C 0.000 }
gfCNCPoint2[17395] = {X 201.2091, Y 33.7058, Z -3.0000, A 0.000, B 0.000, C 0.000 }
gfCNCPoint2[17396] = {X 204.2502, Y 39.9879, Z -3.0000, A 0.000, B 0.000, C 0.000 }
gfCNCPoint2[17397] = {X 204.5648, Y 40.8802, Z -3.0000, A 0.000, B 0.000, C 0.000 }
gfCNCPoint2[17398] = {X 204.6737, Y 41.8200, Z -3.0000, A 0.000, B 0.000, C 0.000 }
gfCNCPoint2[17399] = {X 204.5715, Y 42.7606, Z -3.0000, A 0.000, B 0.000, C 0.000 }
gfCNCPoint2[17400] = {X 204.2633, Y 43.6551, Z -3.0000, A 0.000, B 0.000, C 0.000 }
gfCNCPoint2[17401] = {X 203.7643, Y 44.4590, Z -3.0000, A 0.000, B 0.000, C 0.000 }
gfCNCPoint2[17402] = {X 203.0996, Y 45.1323, Z -3.0000, A 0.000, B 0.000, C 0.000 }
gfCNCPoint2[17403] = {X 202.5633, Y 45.5659, Z -3.0000, A 0.000, B 0.000, C 0.000 }
gfCNCPoint2[17404] = {X 201.8655, Y 46.0240, Z -3.0000, A 0.000, B 0.000, C 0.000 }
gfCNCPoint2[17405] = {X 201.0917, Y 46.3370, Z -3.0000, A 0.000, B 0.000, C 0.000 }
gfCNCPoint2[17406] = {X 200.2716, Y 46.4929, Z -3.0000, A 0.000, B 0.000, C 0.000 }
gfCNCPoint2[17407] = {X 199.4369, Y 46.4858, Z -3.0000, A 0.000, B 0.000, C 0.000 }
gfCNCPoint2[17408] = {X 198.6197, Y 46.3157, Z -3.0000, A 0.000, B 0.000, C 0.000 }
gfCNCPoint2[17409] = {X 196.8802, Y 47.2409, Z -3.0000, A 0.000, B 0.000, C 0.000 }
gfCNCPoint2[17410] = {X 195.0812, Y 48.0442, Z -3.0000, A 0.000, B 0.000, C 0.000 }
gfCNCPoint2[17411] = {X 193.2311, Y 48.7218, Z -3.0000, A 0.000, B 0.000, C 0.000 }
gfCNCPoint2[17412] = {X 191.3389, Y 49.2705, Z -3.0000, A 0.000, B 0.000, C 0.000 }
gfCNCPoint2[17413] = {X 189.4027, Y 49.6628, Z -3.0000, A 0.000, B 0.000, C 0.000 }
gfCNCPoint2[17414] = {X 187.4396, Y 49.8843, Z -3.0000, A 0.000, B 0.000, C 0.000 }
gfCNCPoint2[17415] = {X 185.4646, Y 49.9333, Z -3.0000, A 0.000, B 0.000, C 0.000 }
gfCNCPoint2[17416] = {X 183.4929, Y 49.8094, Z -3.0000, A 0.000, B 0.000, C 0.000 }
gfCNCPoint2[17417] = {X 181.5397, Y 49.5135, Z -3.0000, A 0.000, B 0.000, C 0.000 }
gfCNCPoint2[17418] = {X 179.6620, Y 49.0442, Z -3.0000, A 0.000, B 0.000, C 0.000 }
gfCNCPoint2[17419] = {X 177.8500, Y 48.3639, Z -3.0000, A 0.000, B 0.000, C 0.000 }
gfCNCPoint2[17420] = {X 176.1274, Y 47.4815, Z -3.0000, A 0.000, B 0.000, C 0.000 }
gfCNCPoint2[17421] = {X 174.5166, Y 46.4086, Z -3.0000, A 0.000, B 0.000, C 0.000 }
gfCNCPoint2[17422] = {X 173.2911, Y 45.3743, Z -3.0000, A 0.000, B 0.000, C 0.000 }
gfCNCPoint2[17423] = {X 172.2006, Y 44.1986, Z -3.0000, A 0.000, B 0.000, C 0.000 }
gfCNCPoint2[17424] = {X 171.2612, Y 42.8989, Z -3.0000, A 0.000, B 0.000, C 0.000 }
gfCNCPoint2[17425] = {X 170.4870, Y 41.4945, Z -3.0000, A 0.000, B 0.000, C 0.000 }
gfCNCPoint2[17426] = {X 169.8894, Y 40.0064, Z -3.0000, A 0.000, B 0.000, C 0.000 }
gfCNCPoint2[17427] = {X 169.4774, Y 38.4566, Z -3.0000, A 0.000, B 0.000, C 0.000 }
gfCNCPoint2[17428] = {X 169.2569, Y 36.8682, Z -3.0000, A 0.000, B 0.000, C 0.000 }
gfCNCPoint2[17429] = {X 169.1731, Y 35.0440, Z -3.0000, A 0.000, B 0.000, C 0.000 }
gfCNCPoint2[17430] = {X 169.3184, Y 33.2236, Z -3.0000, A 0.000, B 0.000, C 0.000 }
gfCNCPoint2[17431] = {X 169.6905, Y 31.4357, Z -3.0000, A 0.000, B 0.000, C 0.000 }
gfCNCPoint2[17432] = {X 170.2836, Y 29.7085, Z -3.0000, A 0.000, B 0.000, C 0.000 }
gfCNCPoint2[17433] = {X 170.9356, Y 28.3802, Z -3.0000, A 0.000, B 0.000, C 0.000 }
gfCNCPoint2[17434] = {X 171.7634, Y 27.1537, Z -3.0000, A 0.000, B 0.000, C 0.000 }
gfCNCPoint2[17435] = {X 172.7513, Y 26.0521, Z -3.0000, A 0.000, B 0.000, C 0.000 }
gfCNCPoint2[17436] = {X 173.8807, Y 25.0961, Z -3.0000, A 0.000, B 0.000, C 0.000 }
gfCNCPoint2[17437] = {X 175.1304, Y 24.3038, Z -3.0000, A 0.000, B 0.000, C 0.000 }
gfCNCPoint2[17438] = {X 174.3088, Y 23.9336, Z -3.0000, A 0.000, B 0.000, C 0.000 }
gfCNCPoint2[17439] = {X 173.5839, Y 23.3982, Z -3.0000, A 0.000, B 0.000, C 0.000 }
gfCNCPoint2[17440] = {X 172.9886, Y 22.7217, Z -3.0000, A 0.000, B 0.000, C 0.000 }
gfCNCPoint2[17441] = {X 172.5496, Y 21.9347, Z -3.0000, A 0.000, B 0.000, C 0.000 }
gfCNCPoint2[17442] = {X 171.2322, Y 18.7085, Z -3.0000, A 0.000, B 0.000, C 0.000 }
gfCNCPoint2[17443] = {X 167.5291, Y 20.2207, Z -3.0000, A 0.000, B 0.000, C 0.000 }
gfCNCPoint2[17444] = {X 171.3062, Y 18.6783, Z -3.0000, A 0.000, B 0.000, C 0.000 }
gfCNCPoint2[17445] = {X 169.9886, Y 15.4516, Z -3.0000, A 0.000, B 0.000, C 0.000 }
gfCNCPoint2[17446] = {X 169.7252, Y 14.4911, Z -3.0000, A 0.000, B 0.000, C 0.000 }
gfCNCPoint2[17447] = {X 169.6977, Y 13.4955, Z -3.0000, A 0.000, B 0.000, C 0.000 }
gfCNCPoint2[17448] = {X 169.9076, Y 12.5218, Z -3.0000, A 0.000, B 0.000, C 0.000 }
gfCNCPoint2[17449] = {X 170.3429, Y 11.6260, Z -3.0000, A 0.000, B 0.000, C 0.000 }
gfCNCPoint2[17450] = {X 170.9787, Y 10.8594, Z -3.0000, A 0.000, B 0.000, C 0.000 }
gfCNCPoint2[17451] = {X 171.7785, Y 10.2658, Z -3.0000, A 0.000, B 0.000, C 0.000 }
gfCNCPoint2[17452] = {X 172.4082, Y 9.9068, Z -3.0000, A 0.000, B 0.000, C 0.000 }
gfCNCPoint2[17453] = {X 173.2740, Y 9.5443, Z -3.0000, A 0.000, B 0.000, C 0.000 }
gfCNCPoint2[17454] = {X 174.1991, Y 9.3853, Z -3.0000, A 0.000, B 0.000, C 0.000 }
gfCNCPoint2[17455] = {X 175.1362, Y 9.4376, Z -3.0000, A 0.000, B 0.000, C 0.000 }
gfCNCPoint2[17456] = {X 176.0378, Y 9.6988, Z -3.0000, A 0.000, B 0.000, C 0.000 }
gfCNCPoint2[17457] = {X 178.2241, Y 8.7718, Z -3.0000, A 0.000, B 0.000, C 0.000 }
gfCNCPoint2[17458] = {X 180.4924, Y 8.0693, Z -3.0000, A 0.000, B 0.000, C 0.000 }
gfCNCPoint2[17459] = {X 182.8199, Y 7.5983, Z -3.0000, A 0.000, B 0.000, C 0.000 }
gfCNCPoint2[17460] = {X 185.1830, Y 7.3636, Z -3.0000, A 0.000, B 0.000, C 0.000 }
gfCNCPoint2[17461] = {X 187.5577, Y 7.3677, Z -3.0000, A 0.000, B 0.000, C 0.000 }
gfCNCPoint2[17462] = {X 189.9199, Y 7.6104, Z -3.0000, A 0.000, B 0.000, C 0.000 }
gfCNCPoint2[17463] = {X 191.6611, Y 7.9686, Z -3.0000, A 0.000, B 0.000, C 0.000 }
gfCNCPoint2[17464] = {X 193.3563, Y 8.5036, Z -3.0000, A 0.000, B 0.000, C 0.000 }
gfCNCPoint2[17465] = {X 194.9876, Y 9.2099, Z -3.0000, A 0.000, B 0.000, C 0.000 }
gfCNCPoint2[17466] = {X 196.5378, Y 10.0798, Z -3.0000, A 0.000, B 0.000, C 0.000 }
gfCNCPoint2[17467] = {X 197.9905, Y 11.1044, Z -3.0000, A 0.000, B 0.000, C 0.000 }
gfCNCPoint2[17468] = {X 199.2820, Y 12.2863, Z -3.0000, A 0.000, B 0.000, C 0.000 }
gfCNCPoint2[17469] = {X 200.4014, Y 13.6322, Z -3.0000, A 0.000, B 0.000, C 0.000 }
gfCNCPoint2[17470] = {X 201.3281, Y 15.1175, Z -3.0000, A 0.000, B 0.000, C 0.000 }
gfCNCPoint2[17471] = {X 202.0450, Y 16.7146, Z -3.0000, A 0.000, B 0.000, C 0.000 }
gfCNCPoint2[17472] = {X 202.5139, Y 18.3531, Z -3.0000, A 0.000, B 0.000, C 0.000 }
gfCNCPoint2[17473] = {X 202.7921, Y 20.0344, Z -3.0000, A 0.000, B 0.000, C 0.000 }
gfCNCPoint2[17474] = {X 202.8760, Y 21.7366, Z -3.0000, A 0.000, B 0.000, C 0.000 }
gfCNCPoint2[17475] = {X 202.7646, Y 23.4372, Z -3.0000, A 0.000, B 0.000, C 0.000 }
gfCNCPoint2[17476] = {X 202.4592, Y 25.1138, Z -3.0000, A 0.000, B 0.000, C 0.000 }
gfCNCPoint2[17477] = {X 202.0013, Y 26.5985, Z -3.0000, A 0.000, B 0.000, C 0.000 }
gfCNCPoint2[17478] = {X 201.3480, Y 28.0081, Z -3.0000, A 0.000, B 0.000, C 0.000 }
gfCNCPoint2[17479] = {X 200.5111, Y 29.3171, Z -3.0000, A 0.000, B 0.000, C 0.000 }
gfCNCPoint2[17480] = {X 199.5059, Y 30.5018, Z -3.0000, A 0.000, B 0.000, C 0.000 }
gfCNCPoint2[17481] = {X 198.3505, Y 31.5405, Z -3.0000, A 0.000, B 0.000, C 0.000 }
gfCNCPoint2[17482] = {X 199.2142, Y 31.8438, Z -3.0000, A 0.000, B 0.000, C 0.000 }
gfCNCPoint2[17483] = {X 199.9907, Y 32.3286, Z -3.0000, A 0.000, B 0.000, C 0.000 }
gfCNCPoint2[17484] = {X 200.6423, Y 32.9715, Z -3.0000, A 0.000, B 0.000, C 0.000 }
gfCNCPoint2[17485] = {X 201.1375, Y 33.7414, Z -3.0000, A 0.000, B 0.000, C 0.000 }
gfCNCPoint2[17486] = {X 204.1781, Y 40.0227, Z -3.0000, A 0.000, B 0.000, C 0.000 }
gfCNCPoint2[17487] = {X 204.4868, Y 40.8982, Z -3.0000, A 0.000, B 0.000, C 0.000 }
gfCNCPoint2[17488] = {X 204.5937, Y 41.8203, Z -3.0000, A 0.000, B 0.000, C 0.000 }
gfCNCPoint2[17489] = {X 204.4934, Y 42.7431, Z -3.0000, A 0.000, B 0.000, C 0.000 }
gfCNCPoint2[17490] = {X 204.1910, Y 43.6208, Z -3.0000, A 0.000, B 0.000, C 0.000 }
gfCNCPoint2[17491] = {X 203.7015, Y 44.4095, Z -3.0000, A 0.000, B 0.000, C 0.000 }
gfCNCPoint2[17492] = {X 203.0493, Y 45.0700, Z -3.0000, A 0.000, B 0.000, C 0.000 }
gfCNCPoint2[17493] = {X 202.5130, Y 45.5036, Z -3.0000, A 0.000, B 0.000, C 0.000 }
gfCNCPoint2[17494] = {X 201.8222, Y 45.9563, Z -3.0000, A 0.000, B 0.000, C 0.000 }
gfCNCPoint2[17495] = {X 201.0557, Y 46.2642, Z -3.0000, A 0.000, B 0.000, C 0.000 }
gfCNCPoint2[17496] = {X 200.2436, Y 46.4151, Z -3.0000, A 0.000, B 0.000, C 0.000 }
gfCNCPoint2[17497] = {X 199.4176, Y 46.4031, Z -3.0000, A 0.000, B 0.000, C 0.000 }
gfCNCPoint2[17498] = {X 198.6102, Y 46.2288, Z -3.0000, A 0.000, B 0.000, C 0.000 }
gfCNCPoint2[17499] = {X 196.8688, Y 47.1574, Z -3.0000, A 0.000, B 0.000, C 0.000 }
gfCNCPoint2[17500] = {X 195.0674, Y 47.9635, Z -3.0000, A 0.000, B 0.000, C 0.000 }
gfCNCPoint2[17501] = {X 193.2146, Y 48.6431, Z -3.0000, A 0.000, B 0.000, C 0.000 }
gfCNCPoint2[17502] = {X 191.3193, Y 49.1930, Z -3.0000, A 0.000, B 0.000, C 0.000 }
gfCNCPoint2[17503] = {X 189.3899, Y 49.5838, Z -3.0000, A 0.000, B 0.000, C 0.000 }
gfCNCPoint2[17504] = {X 187.4338, Y 49.8045, Z -3.0000, A 0.000, B 0.000, C 0.000 }
gfCNCPoint2[17505] = {X 185.4658, Y 49.8533, Z -3.0000, A 0.000, B 0.000, C 0.000 }
gfCNCPoint2[17506] = {X 183.5012, Y 49.7298, Z -3.0000, A 0.000, B 0.000, C 0.000 }
gfCNCPoint2[17507] = {X 181.5549, Y 49.4350, Z -3.0000, A 0.000, B 0.000, C 0.000 }
gfCNCPoint2[17508] = {X 179.6859, Y 48.9678, Z -3.0000, A 0.000, B 0.000, C 0.000 }
gfCNCPoint2[17509] = {X 177.8824, Y 48.2907, Z -3.0000, A 0.000, B 0.000, C 0.000 }
gfCNCPoint2[17510] = {X 176.1678, Y 47.4125, Z -3.0000, A 0.000, B 0.000, C 0.000 }
gfCNCPoint2[17511] = {X 174.5645, Y 46.3446, Z -3.0000, A 0.000, B 0.000, C 0.000 }
gfCNCPoint2[17512] = {X 173.3463, Y 45.3164, Z -3.0000, A 0.000, B 0.000, C 0.000 }
gfCNCPoint2[17513] = {X 172.2623, Y 44.1477, Z -3.0000, A 0.000, B 0.000, C 0.000 }
gfCNCPoint2[17514] = {X 171.3286, Y 42.8557, Z -3.0000, A 0.000, B 0.000, C 0.000 }
gfCNCPoint2[17515] = {X 170.5590, Y 41.4597, Z -3.0000, A 0.000, B 0.000, C 0.000 }
gfCNCPoint2[17516] = {X 169.9651, Y 39.9804, Z -3.0000, A 0.000, B 0.000, C 0.000 }
gfCNCPoint2[17517] = {X 169.5556, Y 38.4398, Z -3.0000, A 0.000, B 0.000, C 0.000 }
gfCNCPoint2[17518] = {X 169.3366, Y 36.8608, Z -3.0000, A 0.000, B 0.000, C 0.000 }
gfCNCPoint2[17519] = {X 169.2531, Y 35.0462, Z -3.0000, A 0.000, B 0.000, C 0.000 }
gfCNCPoint2[17520] = {X 169.3975, Y 33.2354, Z -3.0000, A 0.000, B 0.000, C 0.000 }
gfCNCPoint2[17521] = {X 169.7676, Y 31.4570, Z -3.0000, A 0.000, B 0.000, C 0.000 }
gfCNCPoint2[17522] = {X 170.3575, Y 29.7389, Z -3.0000, A 0.000, B 0.000, C 0.000 }
gfCNCPoint2[17523] = {X 171.0242, Y 28.3870, Z -3.0000, A 0.000, B 0.000, C 0.000 }
gfCNCPoint2[17524] = {X 171.8742, Y 27.1421, Z -3.0000, A 0.000, B 0.000, C 0.000 }
gfCNCPoint2[17525] = {X 172.8907, Y 26.0290, Z -3.0000, A 0.000, B 0.000, C 0.000 }
gfCNCPoint2[17526] = {X 174.0535, Y 25.0698, Z -3.0000, A 0.000, B 0.000, C 0.000 }
gfCNCPoint2[17527] = {X 175.3396, Y 24.2834, Z -3.0000, A 0.000, B 0.000, C 0.000 }
gfCNCPoint2[17528] = {X 174.4751, Y 23.9354, Z -3.0000, A 0.000, B 0.000, C 0.000 }
gfCNCPoint2[17529] = {X 173.7099, Y 23.4037, Z -3.0000, A 0.000, B 0.000, C 0.000 }
gfCNCPoint2[17530] = {X 173.0821, Y 22.7150, Z -3.0000, A 0.000, B 0.000, C 0.000 }
gfCNCPoint2[17531] = {X 172.6235, Y 21.9039, Z -3.0000, A 0.000, B 0.000, C 0.000 }
gfCNCPoint2[17532] = {X 171.3062, Y 18.6783, Z -3.0000, A 0.000, B 0.000, C 0.000 }
gfCNCPoint2[17533] = {X 167.6031, Y 20.1905, Z -3.0000, A 0.000, B 0.000, C 0.000 }
gfCNCPoint2[17534] = {X 171.3803, Y 18.6480, Z -3.0000, A 0.000, B 0.000, C 0.000 }
gfCNCPoint2[17535] = {X 170.0626, Y 15.4213, Z -3.0000, A 0.000, B 0.000, C 0.000 }
gfCNCPoint2[17536] = {X 169.8043, Y 14.4793, Z -3.0000, A 0.000, B 0.000, C 0.000 }
gfCNCPoint2[17537] = {X 169.7773, Y 13.5028, Z -3.0000, A 0.000, B 0.000, C 0.000 }
gfCNCPoint2[17538] = {X 169.9832, Y 12.5479, Z -3.0000, A 0.000, B 0.000, C 0.000 }
gfCNCPoint2[17539] = {X 170.4102, Y 11.6694, Z -3.0000, A 0.000, B 0.000, C 0.000 }
gfCNCPoint2[17540] = {X 171.0337, Y 10.9174, Z -3.0000, A 0.000, B 0.000, C 0.000 }
gfCNCPoint2[17541] = {X 171.8181, Y 10.3353, Z -3.0000, A 0.000, B 0.000, C 0.000 }
gfCNCPoint2[17542] = {X 172.4475, Y 9.9764, Z -3.0000, A 0.000, B 0.000, C 0.000 }
gfCNCPoint2[17543] = {X 173.3053, Y 9.6186, Z -3.0000, A 0.000, B 0.000, C 0.000 }
gfCNCPoint2[17544] = {X 174.2218, Y 9.4641, Z -3.0000, A 0.000, B 0.000, C 0.000 }
gfCNCPoint2[17545] = {X 175.1494, Y 9.5211, Z -3.0000, A 0.000, B 0.000, C 0.000 }
gfCNCPoint2[17546] = {X 176.0401, Y 9.7866, Z -3.0000, A 0.000, B 0.000, C 0.000 }
gfCNCPoint2[17547] = {X 178.2232, Y 8.8573, Z -3.0000, A 0.000, B 0.000, C 0.000 }
gfCNCPoint2[17548] = {X 180.4889, Y 8.1527, Z -3.0000, A 0.000, B 0.000, C 0.000 }
gfCNCPoint2[17549] = {X 182.8140, Y 7.6801, Z -3.0000, A 0.000, B 0.000, C 0.000 }
gfCNCPoint2[17550] = {X 185.1749, Y 7.4441, Z -3.0000, A 0.000, B 0.000, C 0.000 }
gfCNCPoint2[17551] = {X 187.5475, Y 7.4473, Z -3.0000, A 0.000, B 0.000, C 0.000 }
gfCNCPoint2[17552] = {X 189.9078, Y 7.6895, Z -3.0000, A 0.000, B 0.000, C 0.000 }
gfCNCPoint2[17553] = {X 191.6409, Y 8.0460, Z -3.0000, A 0.000, B 0.000, C 0.000 }
gfCNCPoint2[17554] = {X 193.3283, Y 8.5786, Z -3.0000, A 0.000, B 0.000, C 0.000 }
gfCNCPoint2[17555] = {X 194.9521, Y 9.2815, Z -3.0000, A 0.000, B 0.000, C 0.000 }
gfCNCPoint2[17556] = {X 196.4951, Y 10.1475, Z -3.0000, A 0.000, B 0.000, C 0.000 }
gfCNCPoint2[17557] = {X 197.9411, Y 11.1673, Z -3.0000, A 0.000, B 0.000, C 0.000 }
gfCNCPoint2[17558] = {X 199.2243, Y 12.3417, Z -3.0000, A 0.000, B 0.000, C 0.000 }
gfCNCPoint2[17559] = {X 200.3365, Y 13.6791, Z -3.0000, A 0.000, B 0.000, C 0.000 }
gfCNCPoint2[17560] = {X 201.2573, Y 15.1548, Z -3.0000, A 0.000, B 0.000, C 0.000 }
gfCNCPoint2[17561] = {X 201.9697, Y 16.7417, Z -3.0000, A 0.000, B 0.000, C 0.000 }
gfCNCPoint2[17562] = {X 202.4360, Y 18.3712, Z -3.0000, A 0.000, B 0.000, C 0.000 }
gfCNCPoint2[17563] = {X 202.7126, Y 20.0435, Z -3.0000, A 0.000, B 0.000, C 0.000 }
gfCNCPoint2[17564] = {X 202.7960, Y 21.7364, Z -3.0000, A 0.000, B 0.000, C 0.000 }
gfCNCPoint2[17565] = {X 202.6851, Y 23.4277, Z -3.0000, A 0.000, B 0.000, C 0.000 }
gfCNCPoint2[17566] = {X 202.3814, Y 25.0952, Z -3.0000, A 0.000, B 0.000, C 0.000 }
gfCNCPoint2[17567] = {X 201.9142, Y 26.6019, Z -3.0000, A 0.000, B 0.000, C 0.000 }
gfCNCPoint2[17568] = {X 201.2445, Y 28.0301, Z -3.0000, A 0.000, B 0.000, C 0.000 }
gfCNCPoint2[17569] = {X 200.3848, Y 29.3527, Z -3.0000, A 0.000, B 0.000, C 0.000 }
gfCNCPoint2[17570] = {X 199.3515, Y 30.5446, Z -3.0000, A 0.000, B 0.000, C 0.000 }
gfCNCPoint2[17571] = {X 198.1642, Y 31.5833, Z -3.0000, A 0.000, B 0.000, C 0.000 }
gfCNCPoint2[17572] = {X 199.0624, Y 31.8619, Z -3.0000, A 0.000, B 0.000, C 0.000 }
gfCNCPoint2[17573] = {X 199.8729, Y 32.3387, Z -3.0000, A 0.000, B 0.000, C 0.000 }
gfCNCPoint2[17574] = {X 200.5527, Y 32.9885, Z -3.0000, A 0.000, B 0.000, C 0.000 }
gfCNCPoint2[17575] = {X 201.0657, Y 33.7766, Z -3.0000, A 0.000, B 0.000, C 0.000 }
gfCNCPoint2[17576] = {X 204.1061, Y 40.0576, Z -3.0000, A 0.000, B 0.000, C 0.000 }
gfCNCPoint2[17577] = {X 204.4089, Y 40.9162, Z -3.0000, A 0.000, B 0.000, C 0.000 }
gfCNCPoint2[17578] = {X 204.5137, Y 41.8206, Z -3.0000, A 0.000, B 0.000, C 0.000 }
gfCNCPoint2[17579] = {X 204.4154, Y 42.7257, Z -3.0000, A 0.000, B 0.000, C 0.000 }
gfCNCPoint2[17580] = {X 204.1188, Y 43.5864, Z -3.0000, A 0.000, B 0.000, C 0.000 }
gfCNCPoint2[17581] = {X 203.6387, Y 44.3600, Z -3.0000, A 0.000, B 0.000, C 0.000 }
gfCNCPoint2[17582] = {X 202.9990, Y 45.0078, Z -3.0000, A 0.000, B 0.000, C 0.000 }
gfCNCPoint2[17583] = {X 202.4628, Y 45.4414, Z -3.0000, A 0.000, B 0.000, C 0.000 }
gfCNCPoint2[17584] = {X 201.7789, Y 45.8887, Z -3.0000, A 0.000, B 0.000, C 0.000 }
gfCNCPoint2[17585] = {X 201.0197, Y 46.1913, Z -3.0000, A 0.000, B 0.000, C 0.000 }
gfCNCPoint2[17586] = {X 200.2156, Y 46.3371, Z -3.0000, A 0.000, B 0.000, C 0.000 }
gfCNCPoint2[17587] = {X 199.3985, Y 46.3203, Z -3.0000, A 0.000, B 0.000, C 0.000 }
gfCNCPoint2[17588] = {X 198.6011, Y 46.1417, Z -3.0000, A 0.000, B 0.000, C 0.000 }
gfCNCPoint2[17589] = {X 196.8577, Y 47.0738, Z -3.0000, A 0.000, B 0.000, C 0.000 }
gfCNCPoint2[17590] = {X 195.0538, Y 47.8826, Z -3.0000, A 0.000, B 0.000, C 0.000 }
gfCNCPoint2[17591] = {X 193.1982, Y 48.5643, Z -3.0000, A 0.000, B 0.000, C 0.000 }
gfCNCPoint2[17592] = {X 191.2996, Y 49.1154, Z -3.0000, A 0.000, B 0.000, C 0.000 }
gfCNCPoint2[17593] = {X 189.3772, Y 49.5049, Z -3.0000, A 0.000, B 0.000, C 0.000 }
gfCNCPoint2[17594] = {X 187.4280, Y 49.7247, Z -3.0000, A 0.000, B 0.000, C 0.000 }
gfCNCPoint2[17595] = {X 185.4671, Y 49.7733, Z -3.0000, A 0.000, B 0.000, C 0.000 }
gfCNCPoint2[17596] = {X 183.5094, Y 49.6502, Z -3.0000, A 0.000, B 0.000, C 0.000 }
gfCNCPoint2[17597] = {X 181.5701, Y 49.3564, Z -3.0000, A 0.000, B 0.000, C 0.000 }
gfCNCPoint2[17598] = {X 179.7099, Y 48.8915, Z -3.0000, A 0.000, B 0.000, C 0.000 }
gfCNCPoint2[17599] = {X 177.9148, Y 48.2176, Z -3.0000, A 0.000, B 0.000, C 0.000 }
gfCNCPoint2[17600] = {X 176.2083, Y 47.3435, Z -3.0000, A 0.000, B 0.000, C 0.000 }
gfCNCPoint2[17601] = {X 174.6125, Y 46.2806, Z -3.0000, A 0.000, B 0.000, C 0.000 }
gfCNCPoint2[17602] = {X 173.4016, Y 45.2586, Z -3.0000, A 0.000, B 0.000, C 0.000 }
gfCNCPoint2[17603] = {X 172.3240, Y 44.0968, Z -3.0000, A 0.000, B 0.000, C 0.000 }
gfCNCPoint2[17604] = {X 171.3959, Y 42.8125, Z -3.0000, A 0.000, B 0.000, C 0.000 }
gfCNCPoint2[17605] = {X 170.6310, Y 41.4248, Z -3.0000, A 0.000, B 0.000, C 0.000 }
gfCNCPoint2[17606] = {X 170.0407, Y 39.9543, Z -3.0000, A 0.000, B 0.000, C 0.000 }
gfCNCPoint2[17607] = {X 169.6338, Y 38.4229, Z -3.0000, A 0.000, B 0.000, C 0.000 }
gfCNCPoint2[17608] = {X 169.4163, Y 36.8534, Z -3.0000, A 0.000, B 0.000, C 0.000 }
gfCNCPoint2[17609] = {X 169.3330, Y 35.0484, Z -3.0000, A 0.000, B 0.000, C 0.000 }
gfCNCPoint2[17610] = {X 169.4766, Y 33.2473, Z -3.0000, A 0.000, B 0.000, C 0.000 }
gfCNCPoint2[17611] = {X 169.8447, Y 31.4783, Z -3.0000, A 0.000, B 0.000, C 0.000 }
gfCNCPoint2[17612] = {X 170.4315, Y 29.7694, Z -3.0000, A 0.000, B 0.000, C 0.000 }
gfCNCPoint2[17613] = {X 171.1149, Y 28.3906, Z -3.0000, A 0.000, B 0.000, C 0.000 }
gfCNCPoint2[17614] = {X 171.9903, Y 27.1250, Z -3.0000, A 0.000, B 0.000, C 0.000 }
gfCNCPoint2[17615] = {X 173.0394, Y 25.9991, Z -3.0000, A 0.000, B 0.000, C 0.000 }
gfCNCPoint2[17616] = {X 174.2402, Y 25.0367, Z -3.0000, A 0.000, B 0.000, C 0.000 }
gfCNCPoint2[17617] = {X 175.5674, Y 24.2579, Z -3.0000, A 0.000, B 0.000, C 0.000 }
gfCNCPoint2[17618] = {X 174.6552, Y 23.9382, Z -3.0000, A 0.000, B 0.000, C 0.000 }
gfCNCPoint2[17619] = {X 173.8438, Y 23.4128, Z -3.0000, A 0.000, B 0.000, C 0.000 }
gfCNCPoint2[17620] = {X 173.1787, Y 22.7113, Z -3.0000, A 0.000, B 0.000, C 0.000 }
gfCNCPoint2[17621] = {X 172.6973, Y 21.8731, Z -3.0000, A 0.000, B 0.000, C 0.000 }
gfCNCPoint2[17622] = {X 171.3803, Y 18.6480, Z -3.0000, A 0.000, B 0.000, C 0.000 }
gfCNCPoint2[17623] = {X 167.6770, Y 20.1603, Z -3.0000, A 0.000, B 0.000, C 0.000 }
gfCNCPoint2[17624] = {X 167.6769, Y 20.1601, Z -3.0000, A 0.000, B 0.000, C 0.000 }
gfCNCPoint2[17625] = {X 171.4542, Y 18.6179, Z -3.0000, A 0.000, B 0.000, C 0.000 }
gfCNCPoint2[17626] = {X 170.1367, Y 15.3911, Z -3.0000, A 0.000, B 0.000, C 0.000 }
gfCNCPoint2[17627] = {X 169.8835, Y 14.4675, Z -3.0000, A 0.000, B 0.000, C 0.000 }
gfCNCPoint2[17628] = {X 169.8570, Y 13.5102, Z -3.0000, A 0.000, B 0.000, C 0.000 }
gfCNCPoint2[17629] = {X 170.0588, Y 12.5740, Z -3.0000, A 0.000, B 0.000, C 0.000 }
gfCNCPoint2[17630] = {X 170.4774, Y 11.7127, Z -3.0000, A 0.000, B 0.000, C 0.000 }
gfCNCPoint2[17631] = {X 171.0888, Y 10.9755, Z -3.0000, A 0.000, B 0.000, C 0.000 }
gfCNCPoint2[17632] = {X 171.8578, Y 10.4048, Z -3.0000, A 0.000, B 0.000, C 0.000 }
gfCNCPoint2[17633] = {X 172.4867, Y 10.0462, Z -3.0000, A 0.000, B 0.000, C 0.000 }
gfCNCPoint2[17634] = {X 173.3363, Y 9.6929, Z -3.0000, A 0.000, B 0.000, C 0.000 }
gfCNCPoint2[17635] = {X 174.2443, Y 9.5431, Z -3.0000, A 0.000, B 0.000, C 0.000 }
gfCNCPoint2[17636] = {X 175.1624, Y 9.6048, Z -3.0000, A 0.000, B 0.000, C 0.000 }
gfCNCPoint2[17637] = {X 176.0421, Y 9.8746, Z -3.0000, A 0.000, B 0.000, C 0.000 }
gfCNCPoint2[17638] = {X 178.2221, Y 8.9430, Z -3.0000, A 0.000, B 0.000, C 0.000 }
gfCNCPoint2[17639] = {X 180.4851, Y 8.2363, Z -3.0000, A 0.000, B 0.000, C 0.000 }
gfCNCPoint2[17640] = {X 182.8078, Y 7.7619, Z -3.0000, A 0.000, B 0.000, C 0.000 }
gfCNCPoint2[17641] = {X 185.1666, Y 7.5246, Z -3.0000, A 0.000, B 0.000, C 0.000 }
gfCNCPoint2[17642] = {X 187.5374, Y 7.5269, Z -3.0000, A 0.000, B 0.000, C 0.000 }
gfCNCPoint2[17643] = {X 189.8957, Y 7.7686, Z -3.0000, A 0.000, B 0.000, C 0.000 }
gfCNCPoint2[17644] = {X 191.6208, Y 8.1234, Z -3.0000, A 0.000, B 0.000, C 0.000 }
gfCNCPoint2[17645] = {X 193.3003, Y 8.6535, Z -3.0000, A 0.000, B 0.000, C 0.000 }
gfCNCPoint2[17646] = {X 194.9166, Y 9.3532, Z -3.0000, A 0.000, B 0.000, C 0.000 }
gfCNCPoint2[17647] = {X 196.4524, Y 10.2151, Z -3.0000, A 0.000, B 0.000, C 0.000 }
gfCNCPoint2[17648] = {X 197.8917, Y 11.2302, Z -3.0000, A 0.000, B 0.000, C 0.000 }
gfCNCPoint2[17649] = {X 199.1666, Y 12.3971, Z -3.0000, A 0.000, B 0.000, C 0.000 }
gfCNCPoint2[17650] = {X 200.2716, Y 13.7259, Z -3.0000, A 0.000, B 0.000, C 0.000 }
gfCNCPoint2[17651] = {X 201.1865, Y 15.1921, Z -3.0000, A 0.000, B 0.000, C 0.000 }
gfCNCPoint2[17652] = {X 201.8944, Y 16.7687, Z -3.0000, A 0.000, B 0.000, C 0.000 }
gfCNCPoint2[17653] = {X 202.3580, Y 18.3894, Z -3.0000, A 0.000, B 0.000, C 0.000 }
gfCNCPoint2[17654] = {X 202.6331, Y 20.0525, Z -3.0000, A 0.000, B 0.000, C 0.000 }
gfCNCPoint2[17655] = {X 202.7160, Y 21.7361, Z -3.0000, A 0.000, B 0.000, C 0.000 }
gfCNCPoint2[17656] = {X 202.6057, Y 23.4182, Z -3.0000, A 0.000, B 0.000, C 0.000 }
gfCNCPoint2[17657] = {X 202.3036, Y 25.0766, Z -3.0000, A 0.000, B 0.000, C 0.000 }
gfCNCPoint2[17658] = {X 201.8261, Y 26.6077, Z -3.0000, A 0.000, B 0.000, C 0.000 }
gfCNCPoint2[17659] = {X 201.1379, Y 28.0565, Z -3.0000, A 0.000, B 0.000, C 0.000 }
gfCNCPoint2[17660] = {X 200.2528, Y 29.3941, Z -3.0000, A 0.000, B 0.000, C 0.000 }
gfCNCPoint2[17661] = {X 199.1883, Y 30.5938, Z -3.0000, A 0.000, B 0.000, C 0.000 }
gfCNCPoint2[17662] = {X 197.9655, Y 31.6318, Z -3.0000, A 0.000, B 0.000, C 0.000 }
gfCNCPoint2[17663] = {X 198.7275, Y 31.8157, Z -3.0000, A 0.000, B 0.000, C 0.000 }
gfCNCPoint2[17664] = {X 199.4389, Y 32.1447, Z -3.0000, A 0.000, B 0.000, C 0.000 }
gfCNCPoint2[17665] = {X 200.0725, Y 32.6060, Z -3.0000, A 0.000, B 0.000, C 0.000 }
gfCNCPoint2[17666] = {X 200.6040, Y 33.1821, Z -3.0000, A 0.000, B 0.000, C 0.000 }
gfCNCPoint2[17667] = {X 201.0129, Y 33.8507, Z -3.0000, A 0.000, B 0.000, C 0.000 }
gfCNCPoint2[17668] = {X 204.0341, Y 40.0925, Z -3.0000, A 0.000, B 0.000, C 0.000 }
gfCNCPoint2[17669] = {X 204.3309, Y 40.9342, Z -3.0000, A 0.000, B 0.000, C 0.000 }
gfCNCPoint2[17670] = {X 204.4337, Y 41.8209, Z -3.0000, A 0.000, B 0.000, C 0.000 }
gfCNCPoint2[17671] = {X 204.3373, Y 42.7082, Z -3.0000, A 0.000, B 0.000, C 0.000 }
gfCNCPoint2[17672] = {X 204.0465, Y 43.5521, Z -3.0000, A 0.000, B 0.000, C 0.000 }
gfCNCPoint2[17673] = {X 203.5758, Y 44.3105, Z -3.0000, A 0.000, B 0.000, C 0.000 }
gfCNCPoint2[17674] = {X 202.9487, Y 44.9456, Z -3.0000, A 0.000, B 0.000, C 0.000 }
gfCNCPoint2[17675] = {X 202.4125, Y 45.3791, Z -3.0000, A 0.000, B 0.000, C 0.000 }
gfCNCPoint2[17676] = {X 201.7356, Y 45.8210, Z -3.0000, A 0.000, B 0.000, C 0.000 }
gfCNCPoint2[17677] = {X 200.9838, Y 46.1183, Z -3.0000, A 0.000, B 0.000, C 0.000 }
gfCNCPoint2[17678] = {X 200.1878, Y 46.2590, Z -3.0000, A 0.000, B 0.000, C 0.000 }
gfCNCPoint2[17679] = {X 199.3797, Y 46.2374, Z -3.0000, A 0.000, B 0.000, C 0.000 }
gfCNCPoint2[17680] = {X 198.5923, Y 46.0543, Z -3.0000, A 0.000, B 0.000, C 0.000 }
gfCNCPoint2[17681] = {X 196.8469, Y 46.9900, Z -3.0000, A 0.000, B 0.000, C 0.000 }
gfCNCPoint2[17682] = {X 195.0404, Y 47.8017, Z -3.0000, A 0.000, B 0.000, C 0.000 }
gfCNCPoint2[17683] = {X 193.1818, Y 48.4854, Z -3.0000, A 0.000, B 0.000, C 0.000 }
gfCNCPoint2[17684] = {X 191.2800, Y 49.0379, Z -3.0000, A 0.000, B 0.000, C 0.000 }
gfCNCPoint2[17685] = {X 189.3644, Y 49.4259, Z -3.0000, A 0.000, B 0.000, C 0.000 }
gfCNCPoint2[17686] = {X 187.4222, Y 49.6449, Z -3.0000, A 0.000, B 0.000, C 0.000 }
gfCNCPoint2[17687] = {X 185.4683, Y 49.6933, Z -3.0000, A 0.000, B 0.000, C 0.000 }
gfCNCPoint2[17688] = {X 183.5177, Y 49.5706, Z -3.0000, A 0.000, B 0.000, C 0.000 }
gfCNCPoint2[17689] = {X 181.5852, Y 49.2779, Z -3.0000, A 0.000, B 0.000, C 0.000 }
gfCNCPoint2[17690] = {X 179.7338, Y 48.8152, Z -3.0000, A 0.000, B 0.000, C 0.000 }
gfCNCPoint2[17691] = {X 177.9472, Y 48.1444, Z -3.0000, A 0.000, B 0.000, C 0.000 }
gfCNCPoint2[17692] = {X 176.2487, Y 47.2744, Z -3.0000, A 0.000, B 0.000, C 0.000 }
gfCNCPoint2[17693] = {X 174.6604, Y 46.2165, Z -3.0000, A 0.000, B 0.000, C 0.000 }
gfCNCPoint2[17694] = {X 173.4568, Y 45.2007, Z -3.0000, A 0.000, B 0.000, C 0.000 }
gfCNCPoint2[17695] = {X 172.3858, Y 44.0459, Z -3.0000, A 0.000, B 0.000, C 0.000 }
gfCNCPoint2[17696] = {X 171.4633, Y 42.7693, Z -3.0000, A 0.000, B 0.000, C 0.000 }
gfCNCPoint2[17697] = {X 170.7031, Y 41.3899, Z -3.0000, A 0.000, B 0.000, C 0.000 }
gfCNCPoint2[17698] = {X 170.1164, Y 39.9283, Z -3.0000, A 0.000, B 0.000, C 0.000 }
gfCNCPoint2[17699] = {X 169.7120, Y 38.4061, Z -3.0000, A 0.000, B 0.000, C 0.000 }
gfCNCPoint2[17700] = {X 169.4959, Y 36.8460, Z -3.0000, A 0.000, B 0.000, C 0.000 }
gfCNCPoint2[17701] = {X 169.4130, Y 35.0507, Z -3.0000, A 0.000, B 0.000, C 0.000 }
gfCNCPoint2[17702] = {X 169.5557, Y 33.2591, Z -3.0000, A 0.000, B 0.000, C 0.000 }
gfCNCPoint2[17703] = {X 169.9218, Y 31.4996, Z -3.0000, A 0.000, B 0.000, C 0.000 }
gfCNCPoint2[17704] = {X 170.5055, Y 29.7998, Z -3.0000, A 0.000, B 0.000, C 0.000 }
gfCNCPoint2[17705] = {X 171.2084, Y 28.3896, Z -3.0000, A 0.000, B 0.000, C 0.000 }
gfCNCPoint2[17706] = {X 172.1137, Y 27.0999, Z -3.0000, A 0.000, B 0.000, C 0.000 }
gfCNCPoint2[17707] = {X 173.2011, Y 25.9596, Z -3.0000, A 0.000, B 0.000, C 0.000 }
gfCNCPoint2[17708] = {X 174.4463, Y 24.9940, Z -3.0000, A 0.000, B 0.000, C 0.000 }
gfCNCPoint2[17709] = {X 175.8215, Y 24.2249, Z -3.0000, A 0.000, B 0.000, C 0.000 }
gfCNCPoint2[17710] = {X 175.0305, Y 24.0139, Z -3.0000, A 0.000, B 0.000, C 0.000 }
gfCNCPoint2[17711] = {X 174.2990, Y 23.6464, Z -3.0000, A 0.000, B 0.000, C 0.000 }
gfCNCPoint2[17712] = {X 173.6576, Y 23.1376, Z -3.0000, A 0.000, B 0.000, C 0.000 }
gfCNCPoint2[17713] = {X 173.1333, Y 22.5089, Z -3.0000, A 0.000, B 0.000, C 0.000 }
gfCNCPoint2[17714] = {X 172.7479, Y 21.7866, Z -3.0000, A 0.000, B 0.000, C 0.000 }
gfCNCPoint2[17715] = {X 171.4542, Y 18.6179, Z -3.0000, A 0.000, B 0.000, C 0.000 }
gfCNCPoint2[17716] = {X 167.6769, Y 20.1601, Z -3.0000, A 0.000, B 0.000, C 0.000 }
gfCNCPoint2[17717] = {X 167.6769, Y 20.1601, Z 0.0000, A 0.000, B 0.000, C 0.000 }
gfCNCPoint2[17718] = {X 167.6769, Y 20.1601, Z 11.0000, A 0.000, B 0.000, C 0.000 }
gfCNCPoint2[17719] = {X 210.1655, Y 28.5741, Z 11.0000, A 0.000, B 0.000, C 0.000 }
gfCNCPoint2[17720] = {X 210.1655, Y 28.5741, Z 0.0000, A 0.000, B 0.000, C 0.000 }
gfCNCPoint2[17721] = {X 210.1655, Y 28.5741, Z -3.0000, A 0.000, B 0.000, C 0.000 }
gfCNCPoint2[17722] = {X 214.2455, Y 28.5741, Z -3.0000, A 0.000, B 0.000, C 0.000 }
gfCNCPoint2[17723] = {X 214.2455, Y 17.4624, Z -3.0000, A 0.000, B 0.000, C 0.000 }
gfCNCPoint2[17724] = {X 214.2402, Y 16.7693, Z -3.0000, A 0.000, B 0.000, C 0.000 }
gfCNCPoint2[17725] = {X 214.2431, Y 16.2729, Z -3.0000, A 0.000, B 0.000, C 0.000 }
gfCNCPoint2[17726] = {X 213.6050, Y 15.6018, Z -3.0000, A 0.000, B 0.000, C 0.000 }
gfCNCPoint2[17727] = {X 213.1247, Y 14.8100, Z -3.0000, A 0.000, B 0.000, C 0.000 }
gfCNCPoint2[17728] = {X 212.8241, Y 13.9340, Z -3.0000, A 0.000, B 0.000, C 0.000 }
gfCNCPoint2[17729] = {X 212.7172, Y 13.0141, Z -3.0000, A 0.000, B 0.000, C 0.000 }
gfCNCPoint2[17730] = {X 212.7170, Y 12.1868, Z -3.0000, A 0.000, B 0.000, C 0.000 }
gfCNCPoint2[17731] = {X 212.8253, Y 11.2255, Z -3.0000, A 0.000, B 0.000, C 0.000 }
gfCNCPoint2[17732] = {X 213.1448, Y 10.3124, Z -3.0000, A 0.000, B 0.000, C 0.000 }
gfCNCPoint2[17733] = {X 213.6595, Y 9.4933, Z -3.0000, A 0.000, B 0.000, C 0.000 }
gfCNCPoint2[17734] = {X 214.3435, Y 8.8093, Z -3.0000, A 0.000, B 0.000, C 0.000 }
gfCNCPoint2[17735] = {X 215.1626, Y 8.2946, Z -3.0000, A 0.000, B 0.000, C 0.000 }
gfCNCPoint2[17736] = {X 216.0757, Y 7.9751, Z -3.0000, A 0.000, B 0.000, C 0.000 }
gfCNCPoint2[17737] = {X 217.0370, Y 7.8668, Z -3.0000, A 0.000, B 0.000, C 0.000 }
gfCNCPoint2[17738] = {X 223.4805, Y 7.8668, Z -3.0000, A 0.000, B 0.000, C 0.000 }
gfCNCPoint2[17739] = {X 224.4418, Y 7.9751, Z -3.0000, A 0.000, B 0.000, C 0.000 }
gfCNCPoint2[17740] = {X 225.3549, Y 8.2946, Z -3.0000, A 0.000, B 0.000, C 0.000 }
gfCNCPoint2[17741] = {X 226.1740, Y 8.8093, Z -3.0000, A 0.000, B 0.000, C 0.000 }
gfCNCPoint2[17742] = {X 226.8580, Y 9.4933, Z -3.0000, A 0.000, B 0.000, C 0.000 }
gfCNCPoint2[17743] = {X 227.3727, Y 10.3124, Z -3.0000, A 0.000, B 0.000, C 0.000 }
gfCNCPoint2[17744] = {X 227.6922, Y 11.2255, Z -3.0000, A 0.000, B 0.000, C 0.000 }
gfCNCPoint2[17745] = {X 227.8005, Y 12.1868, Z -3.0000, A 0.000, B 0.000, C 0.000 }
gfCNCPoint2[17746] = {X 227.8005, Y 12.9781, Z -3.0000, A 0.000, B 0.000, C 0.000 }
gfCNCPoint2[17747] = {X 227.6991, Y 13.9082, Z -3.0000, A 0.000, B 0.000, C 0.000 }
gfCNCPoint2[17748] = {X 227.3999, Y 14.7947, Z -3.0000, A 0.000, B 0.000, C 0.000 }
gfCNCPoint2[17749] = {X 226.9169, Y 15.5960, Z -3.0000, A 0.000, B 0.000, C 0.000 }
gfCNCPoint2[17750] = {X 226.2726, Y 16.2744, Z -3.0000, A 0.000, B 0.000, C 0.000 }
gfCNCPoint2[17751] = {X 226.2735, Y 40.9154, Z -3.0000, A 0.000, B 0.000, C 0.000 }
gfCNCPoint2[17752] = {X 226.9110, Y 41.5854, Z -3.0000, A 0.000, B 0.000, C 0.000 }
gfCNCPoint2[17753] = {X 227.3913, Y 42.3758, Z -3.0000, A 0.000, B 0.000, C 0.000 }
gfCNCPoint2[17754] = {X 227.6923, Y 43.2503, Z -3.0000, A 0.000, B 0.000, C 0.000 }
gfCNCPoint2[17755] = {X 227.8003, Y 44.1689, Z -3.0000, A 0.000, B 0.000, C 0.000 }
gfCNCPoint2[17756] = {X 227.8005, Y 45.0000, Z -3.0000, A 0.000, B 0.000, C 0.000 }
gfCNCPoint2[17757] = {X 227.6922, Y 45.9613, Z -3.0000, A 0.000, B 0.000, C 0.000 }
gfCNCPoint2[17758] = {X 227.3727, Y 46.8744, Z -3.0000, A 0.000, B 0.000, C 0.000 }
gfCNCPoint2[17759] = {X 226.8580, Y 47.6935, Z -3.0000, A 0.000, B 0.000, C 0.000 }
gfCNCPoint2[17760] = {X 226.1740, Y 48.3775, Z -3.0000, A 0.000, B 0.000, C 0.000 }
gfCNCPoint2[17761] = {X 225.3549, Y 48.8922, Z -3.0000, A 0.000, B 0.000, C 0.000 }
gfCNCPoint2[17762] = {X 224.4418, Y 49.2117, Z -3.0000, A 0.000, B 0.000, C 0.000 }
gfCNCPoint2[17763] = {X 223.4805, Y 49.3200, Z -3.0000, A 0.000, B 0.000, C 0.000 }
gfCNCPoint2[17764] = {X 217.0370, Y 49.3200, Z -3.0000, A 0.000, B 0.000, C 0.000 }
gfCNCPoint2[17765] = {X 216.0805, Y 49.2128, Z -3.0000, A 0.000, B 0.000, C 0.000 }
gfCNCPoint2[17766] = {X 215.1715, Y 48.8964, Z -3.0000, A 0.000, B 0.000, C 0.000 }
gfCNCPoint2[17767] = {X 214.3551, Y 48.3867, Z -3.0000, A 0.000, B 0.000, C 0.000 }
gfCNCPoint2[17768] = {X 213.6718, Y 47.7088, Z -3.0000, A 0.000, B 0.000, C 0.000 }
gfCNCPoint2[17769] = {X 213.1556, Y 46.8965, Z -3.0000, A 0.000, B 0.000, C 0.000 }
gfCNCPoint2[17770] = {X 212.8320, Y 45.9901, Z -3.0000, A 0.000, B 0.000, C 0.000 }
gfCNCPoint2[17771] = {X 212.7172, Y 45.0345, Z -3.0000, A 0.000, B 0.000, C 0.000 }
gfCNCPoint2[17772] = {X 212.7170, Y 44.1980, Z -3.0000, A 0.000, B 0.000, C 0.000 }
gfCNCPoint2[17773] = {X 212.7889, Y 43.4191, Z -3.0000, A 0.000, B 0.000, C 0.000 }
gfCNCPoint2[17774] = {X 213.0022, Y 42.6666, Z -3.0000, A 0.000, B 0.000, C 0.000 }
gfCNCPoint2[17775] = {X 213.3496, Y 41.9658, Z -3.0000, A 0.000, B 0.000, C 0.000 }
gfCNCPoint2[17776] = {X 213.8195, Y 41.3404, Z -3.0000, A 0.000, B 0.000, C 0.000 }
gfCNCPoint2[17777] = {X 214.2412, Y 40.8754, Z -3.0000, A 0.000, B 0.000, C 0.000 }
gfCNCPoint2[17778] = {X 214.2455, Y 40.3062, Z -3.0000, A 0.000, B 0.000, C 0.000 }
gfCNCPoint2[17779] = {X 214.2455, Y 28.5741, Z -3.0000, A 0.000, B 0.000, C 0.000 }
gfCNCPoint2[17780] = {X 210.2455, Y 28.5741, Z -3.0000, A 0.000, B 0.000, C 0.000 }
gfCNCPoint2[17781] = {X 214.3255, Y 28.5741, Z -3.0000, A 0.000, B 0.000, C 0.000 }
gfCNCPoint2[17782] = {X 214.3255, Y 17.4621, Z -3.0000, A 0.000, B 0.000, C 0.000 }
gfCNCPoint2[17783] = {X 214.3202, Y 16.7692, Z -3.0000, A 0.000, B 0.000, C 0.000 }
gfCNCPoint2[17784] = {X 214.3233, Y 16.2359, Z -3.0000, A 0.000, B 0.000, C 0.000 }
gfCNCPoint2[17785] = {X 213.6856, Y 15.5753, Z -3.0000, A 0.000, B 0.000, C 0.000 }
gfCNCPoint2[17786] = {X 213.2051, Y 14.7929, Z -3.0000, A 0.000, B 0.000, C 0.000 }
gfCNCPoint2[17787] = {X 212.9042, Y 13.9254, Z -3.0000, A 0.000, B 0.000, C 0.000 }
gfCNCPoint2[17788] = {X 212.7972, Y 13.0135, Z -3.0000, A 0.000, B 0.000, C 0.000 }
gfCNCPoint2[17789] = {X 212.7970, Y 12.1868, Z -3.0000, A 0.000, B 0.000, C 0.000 }
gfCNCPoint2[17790] = {X 212.9033, Y 11.2433, Z -3.0000, A 0.000, B 0.000, C 0.000 }
gfCNCPoint2[17791] = {X 213.2169, Y 10.3472, Z -3.0000, A 0.000, B 0.000, C 0.000 }
gfCNCPoint2[17792] = {X 213.7220, Y 9.5432, Z -3.0000, A 0.000, B 0.000, C 0.000 }
gfCNCPoint2[17793] = {X 214.3934, Y 8.8719, Z -3.0000, A 0.000, B 0.000, C 0.000 }
gfCNCPoint2[17794] = {X 215.1973, Y 8.3667, Z -3.0000, A 0.000, B 0.000, C 0.000 }
gfCNCPoint2[17795] = {X 216.0935, Y 8.0531, Z -3.0000, A 0.000, B 0.000, C 0.000 }
gfCNCPoint2[17796] = {X 217.0370, Y 7.9468, Z -3.0000, A 0.000, B 0.000, C 0.000 }
gfCNCPoint2[17797] = {X 223.4805, Y 7.9468, Z -3.0000, A 0.000, B 0.000, C 0.000 }
gfCNCPoint2[17798] = {X 224.4240, Y 8.0531, Z -3.0000, A 0.000, B 0.000, C 0.000 }
gfCNCPoint2[17799] = {X 225.3201, Y 8.3667, Z -3.0000, A 0.000, B 0.000, C 0.000 }
gfCNCPoint2[17800] = {X 226.1241, Y 8.8718, Z -3.0000, A 0.000, B 0.000, C 0.000 }
gfCNCPoint2[17801] = {X 226.7954, Y 9.5432, Z -3.0000, A 0.000, B 0.000, C 0.000 }
gfCNCPoint2[17802] = {X 227.3006, Y 10.3471, Z -3.0000, A 0.000, B 0.000, C 0.000 }
gfCNCPoint2[17803] = {X 227.6142, Y 11.2433, Z -3.0000, A 0.000, B 0.000, C 0.000 }
gfCNCPoint2[17804] = {X 227.7205, Y 12.1868, Z -3.0000, A 0.000, B 0.000, C 0.000 }
gfCNCPoint2[17805] = {X 227.7205, Y 12.9781, Z -3.0000, A 0.000, B 0.000, C 0.000 }
gfCNCPoint2[17806] = {X 227.6190, Y 13.9000, Z -3.0000, A 0.000, B 0.000, C 0.000 }
gfCNCPoint2[17807] = {X 227.3195, Y 14.7778, Z -3.0000, A 0.000, B 0.000, C 0.000 }
gfCNCPoint2[17808] = {X 226.8364, Y 15.5695, Z -3.0000, A 0.000, B 0.000, C 0.000 }
gfCNCPoint2[17809] = {X 226.1926, Y 16.2371, Z -3.0000, A 0.000, B 0.000, C 0.000 }
gfCNCPoint2[17810] = {X 226.1935, Y 40.9527, Z -3.0000, A 0.000, B 0.000, C 0.000 }
gfCNCPoint2[17811] = {X 226.8306, Y 41.6121, Z -3.0000, A 0.000, B 0.000, C 0.000 }
gfCNCPoint2[17812] = {X 227.3110, Y 42.3931, Z -3.0000, A 0.000, B 0.000, C 0.000 }
gfCNCPoint2[17813] = {X 227.6123, Y 43.2591, Z -3.0000, A 0.000, B 0.000, C 0.000 }
gfCNCPoint2[17814] = {X 227.7203, Y 44.1697, Z -3.0000, A 0.000, B 0.000, C 0.000 }
gfCNCPoint2[17815] = {X 227.7205, Y 45.0000, Z -3.0000, A 0.000, B 0.000, C 0.000 }
gfCNCPoint2[17816] = {X 227.6142, Y 45.9435, Z -3.0000, A 0.000, B 0.000, C 0.000 }
gfCNCPoint2[17817] = {X 227.3006, Y 46.8397, Z -3.0000, A 0.000, B 0.000, C 0.000 }
gfCNCPoint2[17818] = {X 226.7954, Y 47.6436, Z -3.0000, A 0.000, B 0.000, C 0.000 }
gfCNCPoint2[17819] = {X 226.1241, Y 48.3150, Z -3.0000, A 0.000, B 0.000, C 0.000 }
gfCNCPoint2[17820] = {X 225.3201, Y 48.8201, Z -3.0000, A 0.000, B 0.000, C 0.000 }
gfCNCPoint2[17821] = {X 224.4240, Y 49.1337, Z -3.0000, A 0.000, B 0.000, C 0.000 }
gfCNCPoint2[17822] = {X 223.4805, Y 49.2400, Z -3.0000, A 0.000, B 0.000, C 0.000 }
gfCNCPoint2[17823] = {X 217.0370, Y 49.2400, Z -3.0000, A 0.000, B 0.000, C 0.000 }
gfCNCPoint2[17824] = {X 216.0982, Y 49.1348, Z -3.0000, A 0.000, B 0.000, C 0.000 }
gfCNCPoint2[17825] = {X 215.2061, Y 48.8243, Z -3.0000, A 0.000, B 0.000, C 0.000 }
gfCNCPoint2[17826] = {X 214.4048, Y 48.3240, Z -3.0000, A 0.000, B 0.000, C 0.000 }
gfCNCPoint2[17827] = {X 213.7341, Y 47.6587, Z -3.0000, A 0.000, B 0.000, C 0.000 }
gfCNCPoint2[17828] = {X 213.2275, Y 46.8614, Z -3.0000, A 0.000, B 0.000, C 0.000 }
gfCNCPoint2[17829] = {X 212.9099, Y 45.9717, Z -3.0000, A 0.000, B 0.000, C 0.000 }
gfCNCPoint2[17830] = {X 212.7972, Y 45.0338, Z -3.0000, A 0.000, B 0.000, C 0.000 }
gfCNCPoint2[17831] = {X 212.7970, Y 44.1980, Z -3.0000, A 0.000, B 0.000, C 0.000 }
gfCNCPoint2[17832] = {X 212.8676, Y 43.4338, Z -3.0000, A 0.000, B 0.000, C 0.000 }
gfCNCPoint2[17833] = {X 213.0768, Y 42.6954, Z -3.0000, A 0.000, B 0.000, C 0.000 }
gfCNCPoint2[17834] = {X 213.4178, Y 42.0078, Z -3.0000, A 0.000, B 0.000, C 0.000 }
gfCNCPoint2[17835] = {X 213.8788, Y 41.3942, Z -3.0000, A 0.000, B 0.000, C 0.000 }
gfCNCPoint2[17836] = {X 214.3209, Y 40.9065, Z -3.0000, A 0.000, B 0.000, C 0.000 }
gfCNCPoint2[17837] = {X 214.3255, Y 40.3065, Z -3.0000, A 0.000, B 0.000, C 0.000 }
gfCNCPoint2[17838] = {X 214.3255, Y 28.5741, Z -3.0000, A 0.000, B 0.000, C 0.000 }
gfCNCPoint2[17839] = {X 210.3255, Y 28.5741, Z -3.0000, A 0.000, B 0.000, C 0.000 }
gfCNCPoint2[17840] = {X 214.4055, Y 28.5741, Z -3.0000, A 0.000, B 0.000, C 0.000 }
gfCNCPoint2[17841] = {X 214.4055, Y 17.4617, Z -3.0000, A 0.000, B 0.000, C 0.000 }
gfCNCPoint2[17842] = {X 214.4002, Y 16.7692, Z -3.0000, A 0.000, B 0.000, C 0.000 }
gfCNCPoint2[17843] = {X 214.4036, Y 16.1983, Z -3.0000, A 0.000, B 0.000, C 0.000 }
gfCNCPoint2[17844] = {X 213.7662, Y 15.5485, Z -3.0000, A 0.000, B 0.000, C 0.000 }
gfCNCPoint2[17845] = {X 213.2855, Y 14.7756, Z -3.0000, A 0.000, B 0.000, C 0.000 }
gfCNCPoint2[17846] = {X 212.9843, Y 13.9167, Z -3.0000, A 0.000, B 0.000, C 0.000 }
gfCNCPoint2[17847] = {X 212.8772, Y 13.0128, Z -3.0000, A 0.000, B 0.000, C 0.000 }
gfCNCPoint2[17848] = {X 212.8770, Y 12.1868, Z -3.0000, A 0.000, B 0.000, C 0.000 }
gfCNCPoint2[17849] = {X 212.9813, Y 11.2611, Z -3.0000, A 0.000, B 0.000, C 0.000 }
gfCNCPoint2[17850] = {X 213.2890, Y 10.3819, Z -3.0000, A 0.000, B 0.000, C 0.000 }
gfCNCPoint2[17851] = {X 213.7846, Y 9.5931, Z -3.0000, A 0.000, B 0.000, C 0.000 }
gfCNCPoint2[17852] = {X 214.4433, Y 8.9344, Z -3.0000, A 0.000, B 0.000, C 0.000 }
gfCNCPoint2[17853] = {X 215.2321, Y 8.4388, Z -3.0000, A 0.000, B 0.000, C 0.000 }
gfCNCPoint2[17854] = {X 216.1113, Y 8.1311, Z -3.0000, A 0.000, B 0.000, C 0.000 }
gfCNCPoint2[17855] = {X 217.0370, Y 8.0268, Z -3.0000, A 0.000, B 0.000, C 0.000 }
gfCNCPoint2[17856] = {X 223.4805, Y 8.0268, Z -3.0000, A 0.000, B 0.000, C 0.000 }
gfCNCPoint2[17857] = {X 224.4062, Y 8.1311, Z -3.0000, A 0.000, B 0.000, C 0.000 }
gfCNCPoint2[17858] = {X 225.2854, Y 8.4388, Z -3.0000, A 0.000, B 0.000, C 0.000 }
gfCNCPoint2[17859] = {X 226.0742, Y 8.9344, Z -3.0000, A 0.000, B 0.000, C 0.000 }
gfCNCPoint2[17860] = {X 226.7329, Y 9.5931, Z -3.0000, A 0.000, B 0.000, C 0.000 }
gfCNCPoint2[17861] = {X 227.2285, Y 10.3819, Z -3.0000, A 0.000, B 0.000, C 0.000 }
gfCNCPoint2[17862] = {X 227.5362, Y 11.2611, Z -3.0000, A 0.000, B 0.000, C 0.000 }
gfCNCPoint2[17863] = {X 227.6405, Y 12.1868, Z -3.0000, A 0.000, B 0.000, C 0.000 }
gfCNCPoint2[17864] = {X 227.6405, Y 12.9781, Z -3.0000, A 0.000, B 0.000, C 0.000 }
gfCNCPoint2[17865] = {X 227.5389, Y 13.8917, Z -3.0000, A 0.000, B 0.000, C 0.000 }
gfCNCPoint2[17866] = {X 227.2391, Y 14.7607, Z -3.0000, A 0.000, B 0.000, C 0.000 }
gfCNCPoint2[17867] = {X 226.7559, Y 15.5427, Z -3.0000, A 0.000, B 0.000, C 0.000 }
gfCNCPoint2[17868] = {X 226.1126, Y 16.1994, Z -3.0000, A 0.000, B 0.000, C 0.000 }
gfCNCPoint2[17869] = {X 226.1135, Y 40.9904, Z -3.0000, A 0.000, B 0.000, C 0.000 }
gfCNCPoint2[17870] = {X 226.7502, Y 41.6391, Z -3.0000, A 0.000, B 0.000, C 0.000 }
gfCNCPoint2[17871] = {X 227.2307, Y 42.4106, Z -3.0000, A 0.000, B 0.000, C 0.000 }
gfCNCPoint2[17872] = {X 227.5322, Y 43.2680, Z -3.0000, A 0.000, B 0.000, C 0.000 }
gfCNCPoint2[17873] = {X 227.6403, Y 44.1704, Z -3.0000, A 0.000, B 0.000, C 0.000 }
gfCNCPoint2[17874] = {X 227.6405, Y 45.0000, Z -3.0000, A 0.000, B 0.000, C 0.000 }
gfCNCPoint2[17875] = {X 227.5362, Y 45.9257, Z -3.0000, A 0.000, B 0.000, C 0.000 }
gfCNCPoint2[17876] = {X 227.2285, Y 46.8050, Z -3.0000, A 0.000, B 0.000, C 0.000 }
gfCNCPoint2[17877] = {X 226.7329, Y 47.5937, Z -3.0000, A 0.000, B 0.000, C 0.000 }
gfCNCPoint2[17878] = {X 226.0742, Y 48.2524, Z -3.0000, A 0.000, B 0.000, C 0.000 }
gfCNCPoint2[17879] = {X 225.2854, Y 48.7480, Z -3.0000, A 0.000, B 0.000, C 0.000 }
gfCNCPoint2[17880] = {X 224.4062, Y 49.0557, Z -3.0000, A 0.000, B 0.000, C 0.000 }
gfCNCPoint2[17881] = {X 223.4805, Y 49.1600, Z -3.0000, A 0.000, B 0.000, C 0.000 }
gfCNCPoint2[17882] = {X 217.0370, Y 49.1600, Z -3.0000, A 0.000, B 0.000, C 0.000 }
gfCNCPoint2[17883] = {X 216.1160, Y 49.0568, Z -3.0000, A 0.000, B 0.000, C 0.000 }
gfCNCPoint2[17884] = {X 215.2406, Y 48.7521, Z -3.0000, A 0.000, B 0.000, C 0.000 }
gfCNCPoint2[17885] = {X 214.4544, Y 48.2613, Z -3.0000, A 0.000, B 0.000, C 0.000 }
gfCNCPoint2[17886] = {X 213.7965, Y 47.6085, Z -3.0000, A 0.000, B 0.000, C 0.000 }
gfCNCPoint2[17887] = {X 213.2993, Y 46.8263, Z -3.0000, A 0.000, B 0.000, C 0.000 }
gfCNCPoint2[17888] = {X 212.9877, Y 45.9534, Z -3.0000, A 0.000, B 0.000, C 0.000 }
gfCNCPoint2[17889] = {X 212.8771, Y 45.0332, Z -3.0000, A 0.000, B 0.000, C 0.000 }
gfCNCPoint2[17890] = {X 212.8770, Y 44.1980, Z -3.0000, A 0.000, B 0.000, C 0.000 }
gfCNCPoint2[17891] = {X 212.9462, Y 43.4484, Z -3.0000, A 0.000, B 0.000, C 0.000 }
gfCNCPoint2[17892] = {X 213.1515, Y 42.7242, Z -3.0000, A 0.000, B 0.000, C 0.000 }
gfCNCPoint2[17893] = {X 213.4859, Y 42.0497, Z -3.0000, A 0.000, B 0.000, C 0.000 }
gfCNCPoint2[17894] = {X 213.9381, Y 41.4479, Z -3.0000, A 0.000, B 0.000, C 0.000 }
gfCNCPoint2[17895] = {X 214.4007, Y 40.9376, Z -3.0000, A 0.000, B 0.000, C 0.000 }
gfCNCPoint2[17896] = {X 214.4055, Y 40.3069, Z -3.0000, A 0.000, B 0.000, C 0.000 }
gfCNCPoint2[17897] = {X 214.4055, Y 28.5741, Z -3.0000, A 0.000, B 0.000, C 0.000 }
gfCNCPoint2[17898] = {X 210.4055, Y 28.5741, Z -3.0000, A 0.000, B 0.000, C 0.000 }
gfCNCPoint2[17899] = {X 214.4855, Y 28.5741, Z -3.0000, A 0.000, B 0.000, C 0.000 }
gfCNCPoint2[17900] = {X 214.4855, Y 17.4614, Z -3.0000, A 0.000, B 0.000, C 0.000 }
gfCNCPoint2[17901] = {X 214.4802, Y 16.7691, Z -3.0000, A 0.000, B 0.000, C 0.000 }
gfCNCPoint2[17902] = {X 214.4838, Y 16.1604, Z -3.0000, A 0.000, B 0.000, C 0.000 }
gfCNCPoint2[17903] = {X 214.4259, Y 16.1131, Z -3.0000, A 0.000, B 0.000, C 0.000 }
gfCNCPoint2[17904] = {X 214.3689, Y 16.0647, Z -3.0000, A 0.000, B 0.000, C 0.000 }
gfCNCPoint2[17905] = {X 213.7782, Y 15.4329, Z -3.0000, A 0.000, B 0.000, C 0.000 }
gfCNCPoint2[17906] = {X 213.3339, Y 14.6907, Z -3.0000, A 0.000, B 0.000, C 0.000 }
gfCNCPoint2[17907] = {X 213.0560, Y 13.8715, Z -3.0000, A 0.000, B 0.000, C 0.000 }
gfCNCPoint2[17908] = {X 212.9572, Y 13.0121, Z -3.0000, A 0.000, B 0.000, C 0.000 }
gfCNCPoint2[17909] = {X 212.9570, Y 12.1868, Z -3.0000, A 0.000, B 0.000, C 0.000 }
gfCNCPoint2[17910] = {X 213.0593, Y 11.2789, Z -3.0000, A 0.000, B 0.000, C 0.000 }
gfCNCPoint2[17911] = {X 213.3611, Y 10.4166, Z -3.0000, A 0.000, B 0.000, C 0.000 }
gfCNCPoint2[17912] = {X 213.8471, Y 9.6430, Z -3.0000, A 0.000, B 0.000, C 0.000 }
gfCNCPoint2[17913] = {X 214.4932, Y 8.9969, Z -3.0000, A 0.000, B 0.000, C 0.000 }
gfCNCPoint2[17914] = {X 215.2668, Y 8.5109, Z -3.0000, A 0.000, B 0.000, C 0.000 }
gfCNCPoint2[17915] = {X 216.1291, Y 8.2091, Z -3.0000, A 0.000, B 0.000, C 0.000 }
gfCNCPoint2[17916] = {X 217.0370, Y 8.1068, Z -3.0000, A 0.000, B 0.000, C 0.000 }
gfCNCPoint2[17917] = {X 223.4805, Y 8.1068, Z -3.0000, A 0.000, B 0.000, C 0.000 }
gfCNCPoint2[17918] = {X 224.3884, Y 8.2091, Z -3.0000, A 0.000, B 0.000, C 0.000 }
gfCNCPoint2[17919] = {X 225.2507, Y 8.5109, Z -3.0000, A 0.000, B 0.000, C 0.000 }
gfCNCPoint2[17920] = {X 226.0243, Y 8.9969, Z -3.0000, A 0.000, B 0.000, C 0.000 }
gfCNCPoint2[17921] = {X 226.6704, Y 9.6430, Z -3.0000, A 0.000, B 0.000, C 0.000 }
gfCNCPoint2[17922] = {X 227.1564, Y 10.4166, Z -3.0000, A 0.000, B 0.000, C 0.000 }
gfCNCPoint2[17923] = {X 227.4582, Y 11.2789, Z -3.0000, A 0.000, B 0.000, C 0.000 }
gfCNCPoint2[17924] = {X 227.5605, Y 12.1868, Z -3.0000, A 0.000, B 0.000, C 0.000 }
gfCNCPoint2[17925] = {X 227.5605, Y 12.9781, Z -3.0000, A 0.000, B 0.000, C 0.000 }
gfCNCPoint2[17926] = {X 227.4588, Y 13.8834, Z -3.0000, A 0.000, B 0.000, C 0.000 }
gfCNCPoint2[17927] = {X 227.1587, Y 14.7435, Z -3.0000, A 0.000, B 0.000, C 0.000 }
gfCNCPoint2[17928] = {X 226.6753, Y 15.5156, Z -3.0000, A 0.000, B 0.000, C 0.000 }
gfCNCPoint2[17929] = {X 226.0326, Y 16.1612, Z -3.0000, A 0.000, B 0.000, C 0.000 }
gfCNCPoint2[17930] = {X 226.0336, Y 41.0285, Z -3.0000, A 0.000, B 0.000, C 0.000 }
gfCNCPoint2[17931] = {X 226.1409, Y 41.1155, Z -3.0000, A 0.000, B 0.000, C 0.000 }
gfCNCPoint2[17932] = {X 226.7342, Y 41.7472, Z -3.0000, A 0.000, B 0.000, C 0.000 }
gfCNCPoint2[17933] = {X 227.1808, Y 42.4900, Z -3.0000, A 0.000, B 0.000, C 0.000 }
gfCNCPoint2[17934] = {X 227.4603, Y 43.3103, Z -3.0000, A 0.000, B 0.000, C 0.000 }
gfCNCPoint2[17935] = {X 227.5603, Y 44.1712, Z -3.0000, A 0.000, B 0.000, C 0.000 }
gfCNCPoint2[17936] = {X 227.5605, Y 45.0000, Z -3.0000, A 0.000, B 0.000, C 0.000 }
gfCNCPoint2[17937] = {X 227.4582, Y 45.9079, Z -3.0000, A 0.000, B 0.000, C 0.000 }
gfCNCPoint2[17938] = {X 227.1564, Y 46.7702, Z -3.0000, A 0.000, B 0.000, C 0.000 }
gfCNCPoint2[17939] = {X 226.6704, Y 47.5438, Z -3.0000, A 0.000, B 0.000, C 0.000 }
gfCNCPoint2[17940] = {X 226.0243, Y 48.1899, Z -3.0000, A 0.000, B 0.000, C 0.000 }
gfCNCPoint2[17941] = {X 225.2507, Y 48.6760, Z -3.0000, A 0.000, B 0.000, C 0.000 }
gfCNCPoint2[17942] = {X 224.3884, Y 48.9777, Z -3.0000, A 0.000, B 0.000, C 0.000 }
gfCNCPoint2[17943] = {X 223.4805, Y 49.0800, Z -3.0000, A 0.000, B 0.000, C 0.000 }
gfCNCPoint2[17944] = {X 217.0370, Y 49.0800, Z -3.0000, A 0.000, B 0.000, C 0.000 }
gfCNCPoint2[17945] = {X 216.1337, Y 48.9787, Z -3.0000, A 0.000, B 0.000, C 0.000 }
gfCNCPoint2[17946] = {X 215.2752, Y 48.6800, Z -3.0000, A 0.000, B 0.000, C 0.000 }
gfCNCPoint2[17947] = {X 214.5041, Y 48.1986, Z -3.0000, A 0.000, B 0.000, C 0.000 }
gfCNCPoint2[17948] = {X 213.8588, Y 47.5584, Z -3.0000, A 0.000, B 0.000, C 0.000 }
gfCNCPoint2[17949] = {X 213.3712, Y 46.7912, Z -3.0000, A 0.000, B 0.000, C 0.000 }
gfCNCPoint2[17950] = {X 213.0656, Y 45.9351, Z -3.0000, A 0.000, B 0.000, C 0.000 }
gfCNCPoint2[17951] = {X 212.9571, Y 45.0325, Z -3.0000, A 0.000, B 0.000, C 0.000 }
gfCNCPoint2[17952] = {X 212.9570, Y 44.1980, Z -3.0000, A 0.000, B 0.000, C 0.000 }
gfCNCPoint2[17953] = {X 213.0249, Y 43.4631, Z -3.0000, A 0.000, B 0.000, C 0.000 }
gfCNCPoint2[17954] = {X 213.2261, Y 42.7530, Z -3.0000, A 0.000, B 0.000, C 0.000 }
gfCNCPoint2[17955] = {X 213.5540, Y 42.0917, Z -3.0000, A 0.000, B 0.000, C 0.000 }
gfCNCPoint2[17956] = {X 213.9973, Y 41.5016, Z -3.0000, A 0.000, B 0.000, C 0.000 }
gfCNCPoint2[17957] = {X 214.4804, Y 40.9687, Z -3.0000, A 0.000, B 0.000, C 0.000 }
gfCNCPoint2[17958] = {X 214.4855, Y 40.3072, Z -3.0000, A 0.000, B 0.000, C 0.000 }
gfCNCPoint2[17959] = {X 214.4855, Y 28.5741, Z -3.0000, A 0.000, B 0.000, C 0.000 }
gfCNCPoint2[17960] = {X 210.4855, Y 28.5741, Z -3.0000, A 0.000, B 0.000, C 0.000 }
gfCNCPoint2[17961] = {X 214.5655, Y 28.5741, Z -3.0000, A 0.000, B 0.000, C 0.000 }
gfCNCPoint2[17962] = {X 214.5655, Y 17.4611, Z -3.0000, A 0.000, B 0.000, C 0.000 }
gfCNCPoint2[17963] = {X 214.5602, Y 16.7687, Z -3.0000, A 0.000, B 0.000, C 0.000 }
gfCNCPoint2[17964] = {X 214.5595, Y 16.1864, Z -3.0000, A 0.000, B 0.000, C 0.000 }
gfCNCPoint2[17965] = {X 214.5756, Y 16.1310, Z -3.0000, A 0.000, B 0.000, C 0.000 }
gfCNCPoint2[17966] = {X 214.4976, Y 16.0686, Z -3.0000, A 0.000, B 0.000, C 0.000 }
gfCNCPoint2[17967] = {X 214.4213, Y 16.0042, Z -3.0000, A 0.000, B 0.000, C 0.000 }
gfCNCPoint2[17968] = {X 213.8370, Y 15.3780, Z -3.0000, A 0.000, B 0.000, C 0.000 }
gfCNCPoint2[17969] = {X 213.3995, Y 14.6419, Z -3.0000, A 0.000, B 0.000, C 0.000 }
gfCNCPoint2[17970] = {X 213.1287, Y 13.8294, Z -3.0000, A 0.000, B 0.000, C 0.000 }
gfCNCPoint2[17971] = {X 213.0370, Y 12.9779, Z -3.0000, A 0.000, B 0.000, C 0.000 }
gfCNCPoint2[17972] = {X 213.0370, Y 12.1868, Z -3.0000, A 0.000, B 0.000, C 0.000 }
gfCNCPoint2[17973] = {X 213.1373, Y 11.2967, Z -3.0000, A 0.000, B 0.000, C 0.000 }
gfCNCPoint2[17974] = {X 213.4331, Y 10.4513, Z -3.0000, A 0.000, B 0.000, C 0.000 }
gfCNCPoint2[17975] = {X 213.9097, Y 9.6929, Z -3.0000, A 0.000, B 0.000, C 0.000 }
gfCNCPoint2[17976] = {X 214.5431, Y 9.0595, Z -3.0000, A 0.000, B 0.000, C 0.000 }
gfCNCPoint2[17977] = {X 215.3015, Y 8.5829, Z -3.0000, A 0.000, B 0.000, C 0.000 }
gfCNCPoint2[17978] = {X 216.1469, Y 8.2871, Z -3.0000, A 0.000, B 0.000, C 0.000 }
gfCNCPoint2[17979] = {X 217.0370, Y 8.1868, Z -3.0000, A 0.000, B 0.000, C 0.000 }
gfCNCPoint2[17980] = {X 223.4805, Y 8.1868, Z -3.0000, A 0.000, B 0.000, C 0.000 }
gfCNCPoint2[17981] = {X 224.3706, Y 8.2871, Z -3.0000, A 0.000, B 0.000, C 0.000 }
gfCNCPoint2[17982] = {X 225.2160, Y 8.5829, Z -3.0000, A 0.000, B 0.000, C 0.000 }
gfCNCPoint2[17983] = {X 225.9744, Y 9.0595, Z -3.0000, A 0.000, B 0.000, C 0.000 }
gfCNCPoint2[17984] = {X 226.6078, Y 9.6929, Z -3.0000, A 0.000, B 0.000, C 0.000 }
gfCNCPoint2[17985] = {X 227.0844, Y 10.4513, Z -3.0000, A 0.000, B 0.000, C 0.000 }
gfCNCPoint2[17986] = {X 227.3802, Y 11.2967, Z -3.0000, A 0.000, B 0.000, C 0.000 }
gfCNCPoint2[17987] = {X 227.4805, Y 12.1868, Z -3.0000, A 0.000, B 0.000, C 0.000 }
gfCNCPoint2[17988] = {X 227.4803, Y 13.0192, Z -3.0000, A 0.000, B 0.000, C 0.000 }
gfCNCPoint2[17989] = {X 227.3716, Y 13.9049, Z -3.0000, A 0.000, B 0.000, C 0.000 }
gfCNCPoint2[17990] = {X 227.0693, Y 14.7446, Z -3.0000, A 0.000, B 0.000, C 0.000 }
gfCNCPoint2[17991] = {X 226.5883, Y 15.4963, Z -3.0000, A 0.000, B 0.000, C 0.000 }
gfCNCPoint2[17992] = {X 225.9526, Y 16.1226, Z -3.0000, A 0.000, B 0.000, C 0.000 }
gfCNCPoint2[17993] = {X 225.9536, Y 41.0667, Z -3.0000, A 0.000, B 0.000, C 0.000 }
gfCNCPoint2[17994] = {X 226.0924, Y 41.1793, Z -3.0000, A 0.000, B 0.000, C 0.000 }
gfCNCPoint2[17995] = {X 226.6782, Y 41.8057, Z -3.0000, A 0.000, B 0.000, C 0.000 }
gfCNCPoint2[17996] = {X 227.1170, Y 42.5426, Z -3.0000, A 0.000, B 0.000, C 0.000 }
gfCNCPoint2[17997] = {X 227.3886, Y 43.3562, Z -3.0000, A 0.000, B 0.000, C 0.000 }
gfCNCPoint2[17998] = {X 227.4805, Y 44.2089, Z -3.0000, A 0.000, B 0.000, C 0.000 }
gfCNCPoint2[17999] = {X 227.4805, Y 45.0000, Z -3.0000, A 0.000, B 0.000, C 0.000 }
gfCNCPoint2[18000] = {X 227.3802, Y 45.8901, Z -3.0000, A 0.000, B 0.000, C 0.000 }
gfCNCPoint2[18001] = {X 227.0844, Y 46.7355, Z -3.0000, A 0.000, B 0.000, C 0.000 }
gfCNCPoint2[18002] = {X 226.6078, Y 47.4940, Z -3.0000, A 0.000, B 0.000, C 0.000 }
gfCNCPoint2[18003] = {X 225.9744, Y 48.1273, Z -3.0000, A 0.000, B 0.000, C 0.000 }
gfCNCPoint2[18004] = {X 225.2160, Y 48.6039, Z -3.0000, A 0.000, B 0.000, C 0.000 }
gfCNCPoint2[18005] = {X 224.3706, Y 48.8997, Z -3.0000, A 0.000, B 0.000, C 0.000 }
gfCNCPoint2[18006] = {X 223.4805, Y 49.0000, Z -3.0000, A 0.000, B 0.000, C 0.000 }
gfCNCPoint2[18007] = {X 217.0370, Y 49.0000, Z -3.0000, A 0.000, B 0.000, C 0.000 }
gfCNCPoint2[18008] = {X 216.1469, Y 48.8997, Z -3.0000, A 0.000, B 0.000, C 0.000 }
gfCNCPoint2[18009] = {X 215.3015, Y 48.6039, Z -3.0000, A 0.000, B 0.000, C 0.000 }
gfCNCPoint2[18010] = {X 214.5430, Y 48.1273, Z -3.0000, A 0.000, B 0.000, C 0.000 }
gfCNCPoint2[18011] = {X 213.9097, Y 47.4939, Z -3.0000, A 0.000, B 0.000, C 0.000 }
gfCNCPoint2[18012] = {X 213.4331, Y 46.7355, Z -3.0000, A 0.000, B 0.000, C 0.000 }
gfCNCPoint2[18013] = {X 213.1373, Y 45.8900, Z -3.0000, A 0.000, B 0.000, C 0.000 }
gfCNCPoint2[18014] = {X 213.0370, Y 45.0000, Z -3.0000, A 0.000, B 0.000, C 0.000 }
gfCNCPoint2[18015] = {X 213.0370, Y 44.1980, Z -3.0000, A 0.000, B 0.000, C 0.000 }
gfCNCPoint2[18016] = {X 213.1550, Y 43.2418, Z -3.0000, A 0.000, B 0.000, C 0.000 }
gfCNCPoint2[18017] = {X 213.5018, Y 42.3430, Z -3.0000, A 0.000, B 0.000, C 0.000 }
gfCNCPoint2[18018] = {X 214.0566, Y 41.5554, Z -3.0000, A 0.000, B 0.000, C 0.000 }
gfCNCPoint2[18019] = {X 214.5602, Y 40.9999, Z -3.0000, A 0.000, B 0.000, C 0.000 }
gfCNCPoint2[18020] = {X 214.5655, Y 40.3075, Z -3.0000, A 0.000, B 0.000, C 0.000 }
gfCNCPoint2[18021] = {X 214.5655, Y 28.5741, Z -3.0000, A 0.000, B 0.000, C 0.000 }
gfCNCPoint2[18022] = {X 210.4855, Y 28.5741, Z -3.0000, A 0.000, B 0.000, C 0.000 }
gfCNCPoint2[18023] = {X 210.4855, Y 28.5741, Z 0.0000, A 0.000, B 0.000, C 0.000 }
gfCNCPoint2[18024] = {X 210.4855, Y 28.5741, Z 11.0000, A 0.000, B 0.000, C 0.000 }
gfCNCPoint2[18025] = {X 273.6033, Y 28.5937, Z 11.0000, A 0.000, B 0.000, C 0.000 }
gfCNCPoint2[18026] = {X 273.6033, Y 28.5937, Z 0.0000, A 0.000, B 0.000, C 0.000 }
gfCNCPoint2[18027] = {X 273.6033, Y 28.5937, Z -3.0000, A 0.000, B 0.000, C 0.000 }
gfCNCPoint2[18028] = {X 269.5233, Y 28.5936, Z -3.0000, A 0.000, B 0.000, C 0.000 }
gfCNCPoint2[18029] = {X 269.5232, Y 40.9130, Z -3.0000, A 0.000, B 0.000, C 0.000 }
gfCNCPoint2[18030] = {X 269.5370, Y 40.9241, Z -3.0000, A 0.000, B 0.000, C 0.000 }
